LIN {X 0,Y 418.229,Z 234.888,A -85,B 0,C 180,E1 -10045.167,E2 -10045.167} C_VEL
LIN {X 0,Y 418.217,Z 234.887,A -85,B 0,C 180,E1 -10047.48,E2 -10047.48} C_VEL
LIN {X 0,Y 418.245,Z 234.887,A -85,B 0,C 180,E1 -10050.903,E2 -10050.903} C_VEL
LIN {X 0,Y 418.249,Z 234.881,A -85,B 0,C 180,E1 -10054.103,E2 -10054.103} C_VEL
LIN {X 0,Y 418.216,Z 234.893,A -85,B 0,C 180,E1 -10057.271,E2 -10057.271} C_VEL
LIN {X 0,Y 418.27,Z 234.878,A -85,B 0,C 180,E1 -10060.372,E2 -10060.372} C_VEL
LIN {X 0,Y 418.307,Z 234.881,A -85,B 0,C 180,E1 -10063.412,E2 -10063.412} C_VEL
LIN {X 0,Y 418.341,Z 234.871,A -85,B 0,C 180,E1 -10067.007,E2 -10067.007} C_VEL
LIN {X 0,Y 418.335,Z 234.872,A -85,B 0,C 180,E1 -10070.336,E2 -10070.336} C_VEL
LIN {X 0,Y 418.445,Z 234.858,A -85,B 0,C 180,E1 -10073.255,E2 -10073.255} C_VEL
LIN {X 0,Y 418.328,Z 234.872,A -85,B 0,C 180,E1 -10075.188,E2 -10075.188} C_VEL
LIN {X 0,Y 418.543,Z 234.852,A -85,B 0,C 180,E1 -10078.082,E2 -10078.082} C_VEL
LIN {X 0,Y 418.47,Z 234.854,A -85,B 0,C 180,E1 -10080.969,E2 -10080.969} C_VEL
LIN {X 0,Y 418.477,Z 234.853,A -85,B 0,C 180,E1 -10082.894,E2 -10082.894} C_VEL
LIN {X 0,Y 418.494,Z 234.853,A -85,B 0,C 180,E1 -10085.789,E2 -10085.789} C_VEL
LIN {X 0,Y 418.38,Z 234.868,A -85,B 0,C 180,E1 -10088.701,E2 -10088.701} C_VEL
LIN {X 0,Y 418.324,Z 234.872,A -85,B 0,C 180,E1 -10091.636,E2 -10091.636} C_VEL
LIN {X 0,Y 418.315,Z 234.881,A -85,B 0,C 180,E1 -10094.602,E2 -10094.602} C_VEL
LIN {X 0,Y 418.296,Z 234.875,A -85,B 0,C 180,E1 -10097.609,E2 -10097.609} C_VEL
LIN {X 0,Y 418.267,Z 234.886,A -85,B 0,C 180,E1 -10100.667,E2 -10100.667} C_VEL
LIN {X 0,Y 418.276,Z 234.878,A -85,B 0,C 180,E1 -10103.787,E2 -10103.787} C_VEL
LIN {X 0,Y 418.227,Z 234.891,A -85,B 0,C 180,E1 -10107.046,E2 -10107.046} C_VEL
LIN {X 0,Y 418.259,Z 234.88,A -85,B 0,C 180,E1 -10110.276,E2 -10110.276} C_VEL
LIN {X 0,Y 418.253,Z 234.883,A -85,B 0,C 180,E1 -10113.682,E2 -10113.682} C_VEL
LIN {X 0,Y 418.259,Z 234.887,A -85,B 0,C 180,E1 -10117.227,E2 -10117.227} C_VEL
LIN {X 0,Y 418.229,Z 234.885,A -85,B 0,C 180,E1 -10120.869,E2 -10120.869} C_VEL
LIN {X 0,Y 418.202,Z 234.893,A -85,B 0,C 180,E1 -10123.727,E2 -10123.727} C_VEL
LIN {X 0,Y 418.207,Z 234.887,A -85,B 0,C 180,E1 -10126.447,E2 -10126.447} C_VEL
LIN {X 0,Y 418.228,Z 234.885,A -85,B 0,C 180,E1 -10129.134,E2 -10129.134} C_VEL
LIN {X 0,Y 418.255,Z 234.88,A -85,B 0,C 180,E1 -10132.776,E2 -10132.776} C_VEL
LIN {X 0,Y 418.258,Z 234.884,A -85,B 0,C 180,E1 -10136.322,E2 -10136.322} C_VEL
LIN {X 0,Y 418.261,Z 234.883,A -85,B 0,C 180,E1 -10139.728,E2 -10139.728} C_VEL
LIN {X 0,Y 418.285,Z 234.885,A -85,B 0,C 180,E1 -10143.29,E2 -10143.29} C_VEL
LIN {X 0,Y 418.328,Z 235.082,A -85,B 0,C 180,E1 -10143.562,E2 -10143.562} C_VEL
LIN {X 0,Y 420.651,Z 247.12,A -85,B 0,C 180,E1 -10146.359,E2 -10146.359} C_VEL
LIN {X 0,Y 420.968,Z 250.295,A -85,B 0,C 180,E1 -10147.061,E2 -10147.061} C_VEL
LIN {X 0,Y 419.806,Z 267.603,A -85,B 0,C 180,E1 -10150.691,E2 -10150.691} C_VEL
LIN {X 0,Y 419.723,Z 269.608,A -85,B 0,C 180,E1 -10151.068,E2 -10151.068} C_VEL
LIN {X 0,Y 421.486,Z 280.526,A -85,B 0,C 180,E1 -10151.383,E2 -10151.383} C_VEL
LIN {X 0,Y 423.53,Z 293.837,A -85,B 0,C 180,E1 -10151.714,E2 -10151.714} C_VEL
LIN {X 0,Y 422.409,Z 377.431,A -85,B 0,C 180,E1 -10153.227,E2 -10153.227} C_VEL
LIN {X 0,Y 422.039,Z 390.51,A -85,B 0,C 180,E1 -10153.647,E2 -10153.647} C_VEL
LIN {X 0,Y 421.453,Z 402.615,A -85,B 0,C 180,E1 -10154.214,E2 -10154.214} C_VEL
LIN {X 0,Y 420.729,Z 414.885,A -85,B 0,C 180,E1 -10154.993,E2 -10154.993} C_VEL
LIN {X 0,Y 419.97,Z 427.124,A -85,B 0,C 180,E1 -10156.014,E2 -10156.014} C_VEL
LIN {X 0,Y 419.288,Z 438.018,A -85,B 0,C 180,E1 -10157.166,E2 -10157.166} C_VEL
LIN {X 0,Y 418.646,Z 447.21,A -85,B 0,C 180,E1 -10158.377,E2 -10158.377} C_VEL
LIN {X 0,Y 418.062,Z 456.167,A -85,B 0,C 180,E1 -10159.832,E2 -10159.832} C_VEL
LIN {X 0,Y 417.663,Z 463.349,A -85,B 0,C 180,E1 -10161.288,E2 -10161.288} C_VEL
LIN {X 0,Y 417.306,Z 469.059,A -85,B 0,C 180,E1 -10162.742,E2 -10162.742} C_VEL
LIN {X 0,Y 417.136,Z 473.548,A -85,B 0,C 180,E1 -10164.197,E2 -10164.197} C_VEL
LIN {X 0,Y 417.122,Z 475.915,A -85,B 0,C 180,E1 -10165.166,E2 -10165.166} C_VEL
LIN {X 0,Y 417.006,Z 477.844,A -85,B 0,C 180,E1 -10166.133,E2 -10166.133} C_VEL
LIN {X 0,Y 416.99,Z 479.33,A -85,B 0,C 180,E1 -10167.1,E2 -10167.1} C_VEL
LIN {X 0,Y 417.037,Z 480.372,A -85,B 0,C 180,E1 -10168.067,E2 -10168.067} C_VEL
LIN {X 0,Y 416.999,Z 481.017,A -85,B 0,C 180,E1 -10169.033,E2 -10169.033} C_VEL
LIN {X 0,Y 416.989,Z 481.272,A -85,B 0,C 180,E1 -10169.998,E2 -10169.998} C_VEL
LIN {X 0,Y 416.999,Z 481.107,A -85,B 0,C 180,E1 -10170.964,E2 -10170.964} C_VEL
LIN {X 0,Y 417.036,Z 480.518,A -85,B 0,C 180,E1 -10171.93,E2 -10171.93} C_VEL
LIN {X 0,Y 417.005,Z 478.156,A -85,B 0,C 180,E1 -10173.864,E2 -10173.864} C_VEL
LIN {X 0,Y 417.163,Z 475.238,A -85,B 0,C 180,E1 -10175.315,E2 -10175.315} C_VEL
LIN {X 0,Y 417.255,Z 471.278,A -85,B 0,C 180,E1 -10176.769,E2 -10176.769} C_VEL
LIN {X 0,Y 417.612,Z 465.193,A -85,B 0,C 180,E1 -10178.466,E2 -10178.466} C_VEL
LIN {X 0,Y 418.022,Z 458.52,A -85,B 0,C 180,E1 -10179.921,E2 -10179.921} C_VEL
LIN {X 0,Y 418.596,Z 450.239,A -85,B 0,C 180,E1 -10181.376,E2 -10181.376} C_VEL
LIN {X 0,Y 419.307,Z 441.768,A -85,B 0,C 180,E1 -10182.583,E2 -10182.583} C_VEL
LIN {X 0,Y 420.041,Z 431.587,A -85,B 0,C 180,E1 -10183.763,E2 -10183.763} C_VEL
LIN {X 0,Y 420.683,Z 420.983,A -85,B 0,C 180,E1 -10184.758,E2 -10184.758} C_VEL
LIN {X 0,Y 421.436,Z 409.695,A -85,B 0,C 180,E1 -10185.597,E2 -10185.597} C_VEL
LIN {X 0,Y 422.138,Z 398.235,A -85,B 0,C 180,E1 -10186.253,E2 -10186.253} C_VEL
LIN {X 0,Y 422.668,Z 385.205,A -85,B 0,C 180,E1 -10186.791,E2 -10186.791} C_VEL
LIN {X 0,Y 423.061,Z 372.908,A -85,B 0,C 180,E1 -10187.117,E2 -10187.117} C_VEL
LIN {X 0,Y 424.16,Z 293.421,A -85,B 0,C 180,E1 -10188.564,E2 -10188.564} C_VEL
LIN {X 0,Y 419.995,Z 269.208,A -85,B 0,C 180,E1 -10189.255,E2 -10189.255} C_VEL
LIN {X 0,Y 420.004,Z 267.48,A -85,B 0,C 180,E1 -10189.55,E2 -10189.55} C_VEL
LIN {X 0,Y 421.06,Z 250.814,A -85,B 0,C 180,E1 -10192.955,E2 -10192.955} C_VEL
LIN {X 0,Y 420.401,Z 245.236,A -85,B 0,C 180,E1 -10194.176,E2 -10194.176} C_VEL
LIN {X 0,Y 418.317,Z 234.989,A -85,B 0,C 180,E1 -10196.569,E2 -10196.569} C_VEL
LIN {X 0,Y 418.275,Z 234.882,A -85,B 0,C 180,E1 -10199.159,E2 -10199.159} C_VEL
LIN {X 0,Y 418.266,Z 234.883,A -85,B 0,C 180,E1 -10202.84,E2 -10202.84} C_VEL
LIN {X 0,Y 418.251,Z 234.888,A -85,B 0,C 180,E1 -10206.234,E2 -10206.234} C_VEL
LIN {X 0,Y 418.206,Z 234.891,A -85,B 0,C 180,E1 -10209.684,E2 -10209.684} C_VEL
LIN {X 0,Y 418.214,Z 234.891,A -85,B 0,C 180,E1 -10212.314,E2 -10212.314} C_VEL
LIN {X 0,Y 418.239,Z 234.883,A -85,B 0,C 180,E1 -10215.104,E2 -10215.104} C_VEL
LIN {X 0,Y 418.222,Z 234.889,A -85,B 0,C 180,E1 -10217.76,E2 -10217.76} C_VEL
LIN {X 0,Y 418.236,Z 234.884,A -85,B 0,C 180,E1 -10221.551,E2 -10221.551} C_VEL
LIN {X 0,Y 418.25,Z 234.884,A -85,B 0,C 180,E1 -10225.153,E2 -10225.153} C_VEL
LIN {X 0,Y 418.244,Z 234.882,A -85,B 0,C 180,E1 -10227.467,E2 -10227.467} C_VEL
LIN {X 0,Y 418.259,Z 234.885,A -85,B 0,C 180,E1 -10230.893,E2 -10230.893} C_VEL
LIN {X 0,Y 418.215,Z 234.883,A -85,B 0,C 180,E1 -10234.087,E2 -10234.087} C_VEL
LIN {X 0,Y 418.221,Z 234.885,A -85,B 0,C 180,E1 -10237.258,E2 -10237.258} C_VEL
LIN {X 0,Y 418.245,Z 234.885,A -85,B 0,C 180,E1 -10240.357,E2 -10240.357} C_VEL
LIN {X 0,Y 418.273,Z 234.879,A -85,B 0,C 180,E1 -10243.397,E2 -10243.397} C_VEL
LIN {X 0,Y 418.337,Z 234.874,A -85,B 0,C 180,E1 -10246.994,E2 -10246.994} C_VEL
LIN {X 0,Y 418.316,Z 234.875,A -85,B 0,C 180,E1 -10250.322,E2 -10250.322} C_VEL
LIN {X 0,Y 418.452,Z 234.861,A -85,B 0,C 180,E1 -10253.242,E2 -10253.242} C_VEL
LIN {X 0,Y 418.306,Z 234.879,A -85,B 0,C 180,E1 -10255.175,E2 -10255.175} C_VEL
LIN {X 0,Y 418.518,Z 234.85,A -85,B 0,C 180,E1 -10258.069,E2 -10258.069} C_VEL
LIN {X 0,Y 418.649,Z 234.832,A -85,B 0,C 180,E1 -10259.994,E2 -10259.994} C_VEL
LIN {X 0,Y 418.48,Z 234.855,A -85,B 0,C 180,E1 -10262.881,E2 -10262.881} C_VEL
LIN {X 0,Y 418.439,Z 234.86,A -85,B 0,C 180,E1 -10266.474,E2 -10266.474} C_VEL
LIN {X 0,Y 418.372,Z 234.869,A -85,B 0,C 180,E1 -10268.689,E2 -10268.689} C_VEL
LIN {X 0,Y 418.307,Z 234.881,A -85,B 0,C 180,E1 -10271.624,E2 -10271.624} C_VEL
LIN {X 0,Y 418.279,Z 234.881,A -85,B 0,C 180,E1 -10274.59,E2 -10274.59} C_VEL
LIN {X 0,Y 418.255,Z 234.884,A -85,B 0,C 180,E1 -10277.597,E2 -10277.597} C_VEL
LIN {X 0,Y 418.244,Z 234.886,A -85,B 0,C 180,E1 -10280.655,E2 -10280.655} C_VEL
LIN {X 0,Y 418.345,Z 235.06,A -85,B 0,C 180,E1 -10281.902,E2 -10281.902} C_VEL
LIN {X 0,Y 420.612,Z 246.343,A -85,B 0,C 180,E1 -10284.419,E2 -10284.419} C_VEL
LIN {X 0,Y 420.097,Z 258.242,A -85,B 0,C 180,E1 -10286.776,E2 -10286.776} C_VEL
LIN {X 0,Y 424.106,Z 279.087,A -85,B 0,C 180,E1 -10287.408,E2 -10287.408} C_VEL
LIN {X 0,Y 424.207,Z 285.864,A -85,B 0,C 180,E1 -10287.544,E2 -10287.544} C_VEL
LIN {X 0,Y 422.969,Z 366.776,A -85,B 0,C 180,E1 -10289.036,E2 -10289.036} C_VEL
LIN {X 0,Y 422.459,Z 380.788,A -85,B 0,C 180,E1 -10289.501,E2 -10289.501} C_VEL
LIN {X 0,Y 421.952,Z 393.509,A -85,B 0,C 180,E1 -10290.137,E2 -10290.137} C_VEL
LIN {X 0,Y 421.204,Z 406.059,A -85,B 0,C 180,E1 -10290.985,E2 -10290.985} C_VEL
LIN {X 0,Y 420.487,Z 416.903,A -85,B 0,C 180,E1 -10291.925,E2 -10291.925} C_VEL
LIN {X 0,Y 419.791,Z 426.126,A -85,B 0,C 180,E1 -10292.911,E2 -10292.911} C_VEL
LIN {X 0,Y 419.091,Z 435.683,A -85,B 0,C 180,E1 -10294.169,E2 -10294.169} C_VEL
LIN {X 0,Y 418.485,Z 443.34,A -85,B 0,C 180,E1 -10295.397,E2 -10295.397} C_VEL
LIN {X 0,Y 417.912,Z 451.314,A -85,B 0,C 180,E1 -10296.978,E2 -10296.978} C_VEL
LIN {X 0,Y 417.525,Z 457.387,A -85,B 0,C 180,E1 -10298.51,E2 -10298.51} C_VEL
LIN {X 0,Y 417.217,Z 462.602,A -85,B 0,C 180,E1 -10300.241,E2 -10300.241} C_VEL
LIN {X 0,Y 417.03,Z 465.647,A -85,B 0,C 180,E1 -10301.601,E2 -10301.601} C_VEL
LIN {X 0,Y 416.878,Z 468.506,A -85,B 0,C 180,E1 -10303.541,E2 -10303.541} C_VEL
LIN {X 0,Y 416.845,Z 469.573,A -85,B 0,C 180,E1 -10305.069,E2 -10305.069} C_VEL
LIN {X 0,Y 416.8,Z 469.657,A -85,B 0,C 180,E1 -10306.46,E2 -10306.46} C_VEL
LIN {X 0,Y 416.838,Z 468.894,A -85,B 0,C 180,E1 -10307.875,E2 -10307.875} C_VEL
LIN {X 0,Y 416.91,Z 467.21,A -85,B 0,C 180,E1 -10309.325,E2 -10309.325} C_VEL
LIN {X 0,Y 417.058,Z 464.506,A -85,B 0,C 180,E1 -10310.805,E2 -10310.805} C_VEL
LIN {X 0,Y 417.231,Z 460.612,A -85,B 0,C 180,E1 -10312.328,E2 -10312.328} C_VEL
LIN {X 0,Y 417.543,Z 455.256,A -85,B 0,C 180,E1 -10313.909,E2 -10313.909} C_VEL
LIN {X 0,Y 418.018,Z 448.556,A -85,B 0,C 180,E1 -10315.452,E2 -10315.452} C_VEL
LIN {X 0,Y 418.492,Z 440.342,A -85,B 0,C 180,E1 -10316.945,E2 -10316.945} C_VEL
LIN {X 0,Y 419.13,Z 431.379,A -85,B 0,C 180,E1 -10318.26,E2 -10318.26} C_VEL
LIN {X 0,Y 419.746,Z 421.55,A -85,B 0,C 180,E1 -10319.433,E2 -10319.433} C_VEL
LIN {X 0,Y 420.458,Z 410.995,A -85,B 0,C 180,E1 -10320.441,E2 -10320.441} C_VEL
LIN {X 0,Y 421.146,Z 398.632,A -85,B 0,C 180,E1 -10321.375,E2 -10321.375} C_VEL
LIN {X 0,Y 421.714,Z 387.532,A -85,B 0,C 180,E1 -10322.017,E2 -10322.017} C_VEL
LIN {X 0,Y 422.155,Z 374.294,A -85,B 0,C 180,E1 -10322.571,E2 -10322.571} C_VEL
LIN {X 0,Y 422.52,Z 360.472,A -85,B 0,C 180,E1 -10322.932,E2 -10322.932} C_VEL
LIN {X 0,Y 423.47,Z 279.209,A -85,B 0,C 180,E1 -10324.385,E2 -10324.385} C_VEL
LIN {X 0,Y 420.91,Z 264.799,A -85,B 0,C 180,E1 -10324.759,E2 -10324.759} C_VEL
LIN {X 0,Y 419.872,Z 261.526,A -85,B 0,C 180,E1 -10324.945,E2 -10324.945} C_VEL
LIN {X 0,Y 418.385,Z 258.162,A -85,B 0,C 180,E1 -10325.342,E2 -10325.342} C_VEL
LIN {X 0,Y 416.377,Z 254.492,A -85,B 0,C 180,E1 -10326.065,E2 -10326.065} C_VEL
LIN {X 0,Y 413.702,Z 248.584,A -85,B 0,C 180,E1 -10327.592,E2 -10327.592} C_VEL
LIN {X 0,Y 413.252,Z 246.492,A -85,B 0,C 180,E1 -10328.11,E2 -10328.11} C_VEL
LIN {X 0,Y 411.256,Z 235.918,A -85,B 0,C 180,E1 -10330.796,E2 -10330.796} C_VEL
LIN {X 0,Y 411.199,Z 235.765,A -85,B 0,C 180,E1 -10334.132,E2 -10334.132} C_VEL
LIN {X 0,Y 411.242,Z 235.755,A -85,B 0,C 180,E1 -10337.166,E2 -10337.166} C_VEL
LIN {X 0,Y 411.237,Z 235.757,A -85,B 0,C 180,E1 -10340.162,E2 -10340.162} C_VEL
LIN {X 0,Y 411.386,Z 235.739,A -85,B 0,C 180,E1 -10343.134,E2 -10343.134} C_VEL
LIN {X 0,Y 411.249,Z 235.758,A -85,B 0,C 180,E1 -10345.1,E2 -10345.1} C_VEL
LIN {X 0,Y 411.441,Z 235.729,A -85,B 0,C 180,E1 -10348.044,E2 -10348.044} C_VEL
LIN {X 0,Y 411.569,Z 235.713,A -85,B 0,C 180,E1 -10350.002,E2 -10350.002} C_VEL
LIN {X 0,Y 411.403,Z 235.74,A -85,B 0,C 180,E1 -10352.939,E2 -10352.939} C_VEL
LIN {X 0,Y 411.419,Z 235.733,A -85,B 0,C 180,E1 -10355.884,E2 -10355.884} C_VEL
LIN {X 0,Y 411.287,Z 235.751,A -85,B 0,C 180,E1 -10358.848,E2 -10358.848} C_VEL
LIN {X 0,Y 411.233,Z 235.758,A -85,B 0,C 180,E1 -10361.836,E2 -10361.836} C_VEL
LIN {X 0,Y 411.197,Z 235.761,A -85,B 0,C 180,E1 -10364.857,E2 -10364.857} C_VEL
LIN {X 0,Y 411.184,Z 235.765,A -85,B 0,C 180,E1 -10367.92,E2 -10367.92} C_VEL
LIN {X 0,Y 411.13,Z 235.769,A -85,B 0,C 180,E1 -10371.039,E2 -10371.039} C_VEL
LIN {X 0,Y 411.165,Z 235.767,A -85,B 0,C 180,E1 -10374.221,E2 -10374.221} C_VEL
LIN {X 0,Y 411.201,Z 235.762,A -85,B 0,C 180,E1 -10377.483,E2 -10377.483} C_VEL
LIN {X 0,Y 411.144,Z 235.767,A -85,B 0,C 180,E1 -10380.853,E2 -10380.853} C_VEL
LIN {X 0,Y 411.153,Z 235.771,A -85,B 0,C 180,E1 -10384.34,E2 -10384.34} C_VEL
LIN {X 0,Y 411.153,Z 235.769,A -85,B 0,C 180,E1 -10387.98,E2 -10387.98} C_VEL
LIN {X 0,Y 411.164,Z 235.764,A -85,B 0,C 180,E1 -10391.243,E2 -10391.243} C_VEL
LIN {X 0,Y 411.19,Z 235.768,A -85,B 0,C 180,E1 -10394.49,E2 -10394.49} C_VEL
LIN {X 0,Y 411.193,Z 235.761,A -85,B 0,C 180,E1 -10397.304,E2 -10397.304} C_VEL
LIN {X 0,Y 411.196,Z 235.767,A -85,B 0,C 180,E1 -10400.785,E2 -10400.785} C_VEL
LIN {X 0,Y 411.168,Z 235.766,A -85,B 0,C 180,E1 -10404.479,E2 -10404.479} C_VEL
LIN {X 0,Y 411.179,Z 235.769,A -85,B 0,C 180,E1 -10406.881,E2 -10406.881} C_VEL
LIN {X 0,Y 411.192,Z 235.763,A -85,B 0,C 180,E1 -10410.656,E2 -10410.656} C_VEL
LIN {X 0,Y 411.217,Z 235.76,A -85,B 0,C 180,E1 -10413.627,E2 -10413.627} C_VEL
LIN {X 0,Y 411.18,Z 235.765,A -85,B 0,C 180,E1 -10416.86,E2 -10416.86} C_VEL
LIN {X 0,Y 411.201,Z 235.76,A -85,B 0,C 180,E1 -10420.059,E2 -10420.059} C_VEL
LIN {X 0,Y 411.254,Z 235.756,A -85,B 0,C 180,E1 -10423.139,E2 -10423.139} C_VEL
LIN {X 0,Y 411.3,Z 235.747,A -85,B 0,C 180,E1 -10426.904,E2 -10426.904} C_VEL
LIN {X 0,Y 411.288,Z 235.751,A -85,B 0,C 180,E1 -10430.168,E2 -10430.168} C_VEL
LIN {X 0,Y 411.393,Z 235.736,A -85,B 0,C 180,E1 -10433.139,E2 -10433.139} C_VEL
LIN {X 0,Y 411.299,Z 235.747,A -85,B 0,C 180,E1 -10435.106,E2 -10435.106} C_VEL
LIN {X 0,Y 411.512,Z 235.728,A -85,B 0,C 180,E1 -10438.049,E2 -10438.049} C_VEL
LIN {X 0,Y 411.435,Z 235.73,A -85,B 0,C 180,E1 -10440.985,E2 -10440.985} C_VEL
LIN {X 0,Y 411.436,Z 235.73,A -85,B 0,C 180,E1 -10442.944,E2 -10442.944} C_VEL
LIN {X 0,Y 411.439,Z 235.733,A -85,B 0,C 180,E1 -10445.889,E2 -10445.889} C_VEL
LIN {X 0,Y 411.321,Z 235.746,A -85,B 0,C 180,E1 -10448.852,E2 -10448.852} C_VEL
LIN {X 0,Y 411.294,Z 235.749,A -85,B 0,C 180,E1 -10451.838,E2 -10451.838} C_VEL
LIN {X 0,Y 411.273,Z 235.754,A -85,B 0,C 180,E1 -10454.858,E2 -10454.858} C_VEL
LIN {X 0,Y 411.262,Z 235.752,A -85,B 0,C 180,E1 -10457.92,E2 -10457.92} C_VEL
LIN {X 0,Y 411.214,Z 235.762,A -85,B 0,C 180,E1 -10461.038,E2 -10461.038} C_VEL
LIN {X 0,Y 411.21,Z 235.759,A -85,B 0,C 180,E1 -10464.222,E2 -10464.222} C_VEL
LIN {X 0,Y 411.166,Z 235.766,A -85,B 0,C 180,E1 -10467.49,E2 -10467.49} C_VEL
LIN {X 0,Y 411.216,Z 235.758,A -85,B 0,C 180,E1 -10469.717,E2 -10469.717} C_VEL
LIN {X 0,Y 411.226,Z 235.764,A -85,B 0,C 180,E1 -10473.159,E2 -10473.159} C_VEL
LIN {X 0,Y 411.213,Z 235.758,A -85,B 0,C 180,E1 -10476.555,E2 -10476.555} C_VEL
LIN {X 0,Y 411.191,Z 235.764,A -85,B 0,C 180,E1 -10479.722,E2 -10479.722} C_VEL
LIN {X 0,Y 411.14,Z 235.77,A -85,B 0,C 180,E1 -10483.143,E2 -10483.143} C_VEL
LIN {X 0,Y 411.177,Z 235.767,A -85,B 0,C 180,E1 -10485.885,E2 -10485.885} C_VEL
LIN {X 0,Y 411.179,Z 235.766,A -85,B 0,C 180,E1 -10489.494,E2 -10489.494} C_VEL
LIN {X 0,Y 411.203,Z 235.764,A -85,B 0,C 180,E1 -10492.026,E2 -10492.026} C_VEL
LIN {X 0,Y 411.219,Z 235.761,A -85,B 0,C 180,E1 -10495.666,E2 -10495.666} C_VEL
LIN {X 0,Y 411.209,Z 235.759,A -85,B 0,C 180,E1 -10499.153,E2 -10499.153} C_VEL
LIN {X 0,Y 411.209,Z 235.766,A -85,B 0,C 180,E1 -10502.517,E2 -10502.517} C_VEL
LIN {X 0,Y 411.259,Z 235.867,A -85,B 0,C 180,E1 -10503.286,E2 -10503.286} C_VEL
LIN {X 0,Y 413.416,Z 246.889,A -85,B 0,C 180,E1 -10505.92,E2 -10505.92} C_VEL
LIN {X 0,Y 413.979,Z 251.745,A -85,B 0,C 180,E1 -10507.015,E2 -10507.015} C_VEL
LIN {X 0,Y 412.791,Z 269.292,A -85,B 0,C 180,E1 -10510.738,E2 -10510.738} C_VEL
LIN {X 0,Y 413.105,Z 272.049,A -85,B 0,C 180,E1 -10510.869,E2 -10510.869} C_VEL
LIN {X 0,Y 416.732,Z 294.503,A -85,B 0,C 180,E1 -10511.448,E2 -10511.448} C_VEL
LIN {X 0,Y 415.576,Z 377.319,A -85,B 0,C 180,E1 -10512.974,E2 -10512.974} C_VEL
LIN {X 0,Y 415.108,Z 391.143,A -85,B 0,C 180,E1 -10513.429,E2 -10513.429} C_VEL
LIN {X 0,Y 414.551,Z 403.062,A -85,B 0,C 180,E1 -10514.007,E2 -10514.007} C_VEL
LIN {X 0,Y 413.841,Z 414.374,A -85,B 0,C 180,E1 -10514.737,E2 -10514.737} C_VEL
LIN {X 0,Y 413.179,Z 425.156,A -85,B 0,C 180,E1 -10515.631,E2 -10515.631} C_VEL
LIN {X 0,Y 412.383,Z 436.605,A -85,B 0,C 180,E1 -10516.823,E2 -10516.823} C_VEL
LIN {X 0,Y 411.789,Z 445.213,A -85,B 0,C 180,E1 -10517.931,E2 -10517.931} C_VEL
LIN {X 0,Y 411.182,Z 453.143,A -85,B 0,C 180,E1 -10519.162,E2 -10519.162} C_VEL
LIN {X 0,Y 410.696,Z 460.873,A -85,B 0,C 180,E1 -10520.642,E2 -10520.642} C_VEL
LIN {X 0,Y 410.363,Z 467.076,A -85,B 0,C 180,E1 -10522.124,E2 -10522.124} C_VEL
LIN {X 0,Y 410.108,Z 472.311,A -85,B 0,C 180,E1 -10523.713,E2 -10523.713} C_VEL
LIN {X 0,Y 410.036,Z 475.758,A -85,B 0,C 180,E1 -10525.082,E2 -10525.082} C_VEL
LIN {X 0,Y 409.926,Z 477.698,A -85,B 0,C 180,E1 -10526.066,E2 -10526.066} C_VEL
LIN {X 0,Y 409.888,Z 479.202,A -85,B 0,C 180,E1 -10527.05,E2 -10527.05} C_VEL
LIN {X 0,Y 409.933,Z 480.252,A -85,B 0,C 180,E1 -10528.033,E2 -10528.033} C_VEL
LIN {X 0,Y 409.926,Z 480.907,A -85,B 0,C 180,E1 -10529.016,E2 -10529.016} C_VEL
LIN {X 0,Y 409.913,Z 481.169,A -85,B 0,C 180,E1 -10529.998,E2 -10529.998} C_VEL
LIN {X 0,Y 409.925,Z 481.02,A -85,B 0,C 180,E1 -10530.981,E2 -10530.981} C_VEL
LIN {X 0,Y 409.933,Z 480.438,A -85,B 0,C 180,E1 -10531.963,E2 -10531.963} C_VEL
LIN {X 0,Y 409.927,Z 478.088,A -85,B 0,C 180,E1 -10533.931,E2 -10533.931} C_VEL
LIN {X 0,Y 410.081,Z 475.183,A -85,B 0,C 180,E1 -10535.407,E2 -10535.407} C_VEL
LIN {X 0,Y 410.193,Z 471.236,A -85,B 0,C 180,E1 -10536.886,E2 -10536.886} C_VEL
LIN {X 0,Y 410.498,Z 466.147,A -85,B 0,C 180,E1 -10538.366,E2 -10538.366} C_VEL
LIN {X 0,Y 410.914,Z 459.751,A -85,B 0,C 180,E1 -10539.846,E2 -10539.846} C_VEL
LIN {X 0,Y 411.502,Z 451.742,A -85,B 0,C 180,E1 -10541.325,E2 -10541.325} C_VEL
LIN {X 0,Y 412.385,Z 441.792,A -85,B 0,C 180,E1 -10542.798,E2 -10542.798} C_VEL
LIN {X 0,Y 413.103,Z 432.283,A -85,B 0,C 180,E1 -10543.931,E2 -10543.931} C_VEL
LIN {X 0,Y 413.83,Z 421.097,A -85,B 0,C 180,E1 -10545.008,E2 -10545.008} C_VEL
LIN {X 0,Y 414.62,Z 409.885,A -85,B 0,C 180,E1 -10545.86,E2 -10545.86} C_VEL
LIN {X 0,Y 415.359,Z 398.557,A -85,B 0,C 180,E1 -10546.525,E2 -10546.525} C_VEL
LIN {X 0,Y 415.908,Z 385.789,A -85,B 0,C 180,E1 -10547.072,E2 -10547.072} C_VEL
LIN {X 0,Y 416.371,Z 372.533,A -85,B 0,C 180,E1 -10547.432,E2 -10547.432} C_VEL
LIN {X 0,Y 417.434,Z 293.78,A -85,B 0,C 180,E1 -10548.898,E2 -10548.898} C_VEL
LIN {X 0,Y 413.326,Z 270.34,A -85,B 0,C 180,E1 -10549.575,E2 -10549.575} C_VEL
LIN {X 0,Y 413.082,Z 268.6,A -85,B 0,C 180,E1 -10549.678,E2 -10549.678} C_VEL
LIN {X 0,Y 414.121,Z 252.699,A -85,B 0,C 180,E1 -10552.973,E2 -10552.973} C_VEL
LIN {X 0,Y 413.941,Z 249.262,A -85,B 0,C 180,E1 -10553.722,E2 -10553.722} C_VEL
LIN {X 0,Y 411.965,Z 239.075,A -85,B 0,C 180,E1 -10556.072,E2 -10556.072} C_VEL
LIN {X 0,Y 411.251,Z 235.81,A -85,B 0,C 180,E1 -10556.917,E2 -10556.917} C_VEL
LIN {X 0,Y 411.21,Z 235.765,A -85,B 0,C 180,E1 -10559.71,E2 -10559.71} C_VEL
LIN {X 0,Y 411.216,Z 235.762,A -85,B 0,C 180,E1 -10563.152,E2 -10563.152} C_VEL
LIN {X 0,Y 411.199,Z 235.764,A -85,B 0,C 180,E1 -10566.548,E2 -10566.548} C_VEL
LIN {X 0,Y 411.175,Z 235.767,A -85,B 0,C 180,E1 -10569.716,E2 -10569.716} C_VEL
LIN {X 0,Y 411.168,Z 235.764,A -85,B 0,C 180,E1 -10573.131,E2 -10573.131} C_VEL
LIN {X 0,Y 411.168,Z 235.766,A -85,B 0,C 180,E1 -10575.878,E2 -10575.878} C_VEL
LIN {X 0,Y 411.161,Z 235.767,A -85,B 0,C 180,E1 -10579.488,E2 -10579.488} C_VEL
LIN {X 0,Y 411.183,Z 235.766,A -85,B 0,C 180,E1 -10582.02,E2 -10582.02} C_VEL
LIN {X 0,Y 411.202,Z 235.762,A -85,B 0,C 180,E1 -10585.119,E2 -10585.119} C_VEL
LIN {X 0,Y 411.164,Z 235.766,A -85,B 0,C 180,E1 -10587.998,E2 -10587.998} C_VEL
LIN {X 0,Y 411.171,Z 235.765,A -85,B 0,C 180,E1 -10591.401,E2 -10591.401} C_VEL
LIN {X 0,Y 411.186,Z 235.767,A -85,B 0,C 180,E1 -10594.936,E2 -10594.936} C_VEL
LIN {X 0,Y 411.195,Z 235.759,A -85,B 0,C 180,E1 -10597.908,E2 -10597.908} C_VEL
LIN {X 0,Y 411.177,Z 235.764,A -85,B 0,C 180,E1 -10601.044,E2 -10601.044} C_VEL
LIN {X 0,Y 411.199,Z 235.759,A -85,B 0,C 180,E1 -10604.124,E2 -10604.124} C_VEL
LIN {X 0,Y 411.294,Z 235.749,A -85,B 0,C 180,E1 -10607.16,E2 -10607.16} C_VEL
LIN {X 0,Y 411.27,Z 235.753,A -85,B 0,C 180,E1 -10610.155,E2 -10610.155} C_VEL
LIN {X 0,Y 411.418,Z 235.738,A -85,B 0,C 180,E1 -10613.126,E2 -10613.126} C_VEL
LIN {X 0,Y 411.279,Z 235.753,A -85,B 0,C 180,E1 -10615.093,E2 -10615.093} C_VEL
LIN {X 0,Y 411.487,Z 235.726,A -85,B 0,C 180,E1 -10618.036,E2 -10618.036} C_VEL
LIN {X 0,Y 411.619,Z 235.708,A -85,B 0,C 180,E1 -10619.994,E2 -10619.994} C_VEL
LIN {X 0,Y 411.437,Z 235.732,A -85,B 0,C 180,E1 -10622.931,E2 -10622.931} C_VEL
LIN {X 0,Y 411.407,Z 235.738,A -85,B 0,C 180,E1 -10626.861,E2 -10626.861} C_VEL
LIN {X 0,Y 411.283,Z 235.755,A -85,B 0,C 180,E1 -10629.832,E2 -10629.832} C_VEL
LIN {X 0,Y 411.286,Z 235.754,A -85,B 0,C 180,E1 -10633.103,E2 -10633.103} C_VEL
LIN {X 0,Y 411.225,Z 235.761,A -85,B 0,C 180,E1 -10636.882,E2 -10636.882} C_VEL
LIN {X 0,Y 411.221,Z 235.764,A -85,B 0,C 180,E1 -10639.979,E2 -10639.979} C_VEL
LIN {X 0,Y 411.254,Z 235.868,A -85,B 0,C 180,E1 -10641.548,E2 -10641.548} C_VEL
LIN {X 0,Y 413.129,Z 244.487,A -85,B 0,C 180,E1 -10643.555,E2 -10643.555} C_VEL
LIN {X 0,Y 413.734,Z 247.939,A -85,B 0,C 180,E1 -10644.317,E2 -10644.317} C_VEL
LIN {X 0,Y 413.234,Z 258.335,A -85,B 0,C 180,E1 -10646.404,E2 -10646.404} C_VEL
LIN {X 0,Y 417.379,Z 279.278,A -85,B 0,C 180,E1 -10647.066,E2 -10647.066} C_VEL
LIN {X 0,Y 417.607,Z 283.906,A -85,B 0,C 180,E1 -10647.169,E2 -10647.169} C_VEL
LIN {X 0,Y 416.24,Z 367.025,A -85,B 0,C 180,E1 -10648.73,E2 -10648.73} C_VEL
LIN {X 0,Y 415.747,Z 380.483,A -85,B 0,C 180,E1 -10649.184,E2 -10649.184} C_VEL
LIN {X 0,Y 415.257,Z 392.681,A -85,B 0,C 180,E1 -10649.792,E2 -10649.792} C_VEL
LIN {X 0,Y 414.517,Z 404.274,A -85,B 0,C 180,E1 -10650.563,E2 -10650.563} C_VEL
LIN {X 0,Y 413.665,Z 416.606,A -85,B 0,C 180,E1 -10651.628,E2 -10651.628} C_VEL
LIN {X 0,Y 412.879,Z 426.512,A -85,B 0,C 180,E1 -10652.704,E2 -10652.704} C_VEL
LIN {X 0,Y 412.104,Z 436.233,A -85,B 0,C 180,E1 -10654.015,E2 -10654.015} C_VEL
LIN {X 0,Y 411.372,Z 445.122,A -85,B 0,C 180,E1 -10655.501,E2 -10655.501} C_VEL
LIN {X 0,Y 410.831,Z 452.573,A -85,B 0,C 180,E1 -10657.075,E2 -10657.075} C_VEL
LIN {X 0,Y 410.439,Z 458.504,A -85,B 0,C 180,E1 -10658.67,E2 -10658.67} C_VEL
LIN {X 0,Y 410.158,Z 462.542,A -85,B 0,C 180,E1 -10660.056,E2 -10660.056} C_VEL
LIN {X 0,Y 410.019,Z 464.852,A -85,B 0,C 180,E1 -10661.049,E2 -10661.049} C_VEL
LIN {X 0,Y 409.868,Z 467.395,A -85,B 0,C 180,E1 -10662.5,E2 -10662.5} C_VEL
LIN {X 0,Y 409.767,Z 468.997,A -85,B 0,C 180,E1 -10663.92,E2 -10663.92} C_VEL
LIN {X 0,Y 409.738,Z 469.752,A -85,B 0,C 180,E1 -10665.315,E2 -10665.315} C_VEL
LIN {X 0,Y 409.707,Z 469.713,A -85,B 0,C 180,E1 -10666.677,E2 -10666.677} C_VEL
LIN {X 0,Y 409.738,Z 468.88,A -85,B 0,C 180,E1 -10668.017,E2 -10668.017} C_VEL
LIN {X 0,Y 409.823,Z 467.336,A -85,B 0,C 180,E1 -10669.336,E2 -10669.336} C_VEL
LIN {X 0,Y 409.953,Z 465.096,A -85,B 0,C 180,E1 -10670.634,E2 -10670.634} C_VEL
LIN {X 0,Y 410.138,Z 461.853,A -85,B 0,C 180,E1 -10672.006,E2 -10672.006} C_VEL
LIN {X 0,Y 410.417,Z 456.973,A -85,B 0,C 180,E1 -10673.577,E2 -10673.577} C_VEL
LIN {X 0,Y 410.82,Z 450.5,A -85,B 0,C 180,E1 -10675.183,E2 -10675.183} C_VEL
LIN {X 0,Y 411.262,Z 443.582,A -85,B 0,C 180,E1 -10676.56,E2 -10676.56} C_VEL
LIN {X 0,Y 411.874,Z 435.171,A -85,B 0,C 180,E1 -10677.923,E2 -10677.923} C_VEL
LIN {X 0,Y 412.586,Z 424.813,A -85,B 0,C 180,E1 -10679.271,E2 -10679.271} C_VEL
LIN {X 0,Y 413.37,Z 413.288,A -85,B 0,C 180,E1 -10680.461,E2 -10680.461} C_VEL
LIN {X 0,Y 414.075,Z 401.402,A -85,B 0,C 180,E1 -10681.42,E2 -10681.42} C_VEL
LIN {X 0,Y 414.781,Z 389.372,A -85,B 0,C 180,E1 -10682.162,E2 -10682.162} C_VEL
LIN {X 0,Y 415.257,Z 376.598,A -85,B 0,C 180,E1 -10682.743,E2 -10682.743} C_VEL
LIN {X 0,Y 415.605,Z 364.099,A -85,B 0,C 180,E1 -10683.113,E2 -10683.113} C_VEL
LIN {X 0,Y 416.683,Z 280.106,A -85,B 0,C 180,E1 -10684.65,E2 -10684.65} C_VEL
LIN {X 0,Y 412.95,Z 259.401,A -85,B 0,C 180,E1 -10685.225,E2 -10685.225} C_VEL
LIN {X 0,Y 412.898,Z 258.328,A -85,B 0,C 180,E1 -10685.356,E2 -10685.356} C_VEL
LIN {X 0,Y 413.503,Z 248.925,A -85,B 0,C 180,E1 -10687.519,E2 -10687.519} C_VEL
LIN {X 0,Y 413.252,Z 246.492,A -85,B 0,C 180,E1 -10688.11,E2 -10688.11} C_VEL
LIN {X 0,Y 412.274,Z 244.732,A -85,B 0,C 180,E1 -10688.584,E2 -10688.584} C_VEL
LIN {X 0,Y 408.926,Z 242.416,A -85,B 0,C 180,E1 -10689.333,E2 -10689.333} C_VEL
LIN {X 0,Y 405.538,Z 240.125,A -85,B 0,C 180,E1 -10690.094,E2 -10690.094} C_VEL
LIN {X 0,Y 404.517,Z 238.393,A -85,B 0,C 180,E1 -10690.583,E2 -10690.583} C_VEL
LIN {X 0,Y 404.156,Z 236.672,A -85,B 0,C 180,E1 -10691.105,E2 -10691.105} C_VEL
LIN {X 0,Y 404.16,Z 236.64,A -85,B 0,C 180,E1 -10693.848,E2 -10693.848} C_VEL
LIN {X 0,Y 404.209,Z 236.633,A -85,B 0,C 180,E1 -10696.938,E2 -10696.938} C_VEL
LIN {X 0,Y 404.2,Z 236.632,A -85,B 0,C 180,E1 -10699.989,E2 -10699.989} C_VEL
LIN {X 0,Y 404.333,Z 236.619,A -85,B 0,C 180,E1 -10703.013,E2 -10703.013} C_VEL
LIN {X 0,Y 404.22,Z 236.634,A -85,B 0,C 180,E1 -10705.015,E2 -10705.015} C_VEL
LIN {X 0,Y 404.411,Z 236.605,A -85,B 0,C 180,E1 -10708.01,E2 -10708.01} C_VEL
LIN {X 0,Y 404.539,Z 236.589,A -85,B 0,C 180,E1 -10710.002,E2 -10710.002} C_VEL
LIN {X 0,Y 404.36,Z 236.618,A -85,B 0,C 180,E1 -10712.991,E2 -10712.991} C_VEL
LIN {X 0,Y 404.365,Z 236.611,A -85,B 0,C 180,E1 -10715.987,E2 -10715.987} C_VEL
LIN {X 0,Y 404.226,Z 236.632,A -85,B 0,C 180,E1 -10719.004,E2 -10719.004} C_VEL
LIN {X 0,Y 404.203,Z 236.632,A -85,B 0,C 180,E1 -10722.045,E2 -10722.045} C_VEL
LIN {X 0,Y 404.142,Z 236.642,A -85,B 0,C 180,E1 -10725.122,E2 -10725.122} C_VEL
LIN {X 0,Y 404.142,Z 236.64,A -85,B 0,C 180,E1 -10728.243,E2 -10728.243} C_VEL
LIN {X 0,Y 404.073,Z 236.651,A -85,B 0,C 180,E1 -10731.424,E2 -10731.424} C_VEL
LIN {X 0,Y 404.116,Z 236.642,A -85,B 0,C 180,E1 -10734.671,E2 -10734.671} C_VEL
LIN {X 0,Y 404.139,Z 236.646,A -85,B 0,C 180,E1 -10738.005,E2 -10738.005} C_VEL
LIN {X 0,Y 404.091,Z 236.647,A -85,B 0,C 180,E1 -10741.566,E2 -10741.566} C_VEL
LIN {X 0,Y 404.132,Z 236.64,A -85,B 0,C 180,E1 -10745.023,E2 -10745.023} C_VEL
LIN {X 0,Y 404.114,Z 236.645,A -85,B 0,C 180,E1 -10748.763,E2 -10748.763} C_VEL
LIN {X 0,Y 404.146,Z 236.638,A -85,B 0,C 180,E1 -10751.618,E2 -10751.618} C_VEL
LIN {X 0,Y 404.155,Z 236.645,A -85,B 0,C 180,E1 -10754.537,E2 -10754.537} C_VEL
LIN {X 0,Y 404.172,Z 236.636,A -85,B 0,C 180,E1 -10757.313,E2 -10757.313} C_VEL
LIN {X 0,Y 404.134,Z 236.64,A -85,B 0,C 180,E1 -10759.963,E2 -10759.963} C_VEL
LIN {X 0,Y 404.108,Z 236.647,A -85,B 0,C 180,E1 -10763.132,E2 -10763.132} C_VEL
LIN {X 0,Y 404.116,Z 236.642,A -85,B 0,C 180,E1 -10766.196,E2 -10766.196} C_VEL
LIN {X 0,Y 404.121,Z 236.642,A -85,B 0,C 180,E1 -10769.723,E2 -10769.723} C_VEL
LIN {X 0,Y 404.175,Z 236.642,A -85,B 0,C 180,E1 -10773.131,E2 -10773.131} C_VEL
LIN {X 0,Y 404.156,Z 236.643,A -85,B 0,C 180,E1 -10775.342,E2 -10775.342} C_VEL
LIN {X 0,Y 404.123,Z 236.641,A -85,B 0,C 180,E1 -10778.588,E2 -10778.588} C_VEL
LIN {X 0,Y 404.193,Z 236.636,A -85,B 0,C 180,E1 -10781.769,E2 -10781.769} C_VEL
LIN {X 0,Y 404.197,Z 236.633,A -85,B 0,C 180,E1 -10784.89,E2 -10784.89} C_VEL
LIN {X 0,Y 404.25,Z 236.629,A -85,B 0,C 180,E1 -10787.966,E2 -10787.966} C_VEL
LIN {X 0,Y 404.264,Z 236.624,A -85,B 0,C 180,E1 -10791.006,E2 -10791.006} C_VEL
LIN {X 0,Y 404.381,Z 236.614,A -85,B 0,C 180,E1 -10794.021,E2 -10794.021} C_VEL
LIN {X 0,Y 404.481,Z 236.604,A -85,B 0,C 180,E1 -10798.015,E2 -10798.015} C_VEL
LIN {X 0,Y 404.401,Z 236.606,A -85,B 0,C 180,E1 -10801.002,E2 -10801.002} C_VEL
LIN {X 0,Y 404.395,Z 236.607,A -85,B 0,C 180,E1 -10802.995,E2 -10802.995} C_VEL
LIN {X 0,Y 404.388,Z 236.612,A -85,B 0,C 180,E1 -10805.992,E2 -10805.992} C_VEL
LIN {X 0,Y 404.27,Z 236.624,A -85,B 0,C 180,E1 -10809.007,E2 -10809.007} C_VEL
LIN {X 0,Y 404.268,Z 236.626,A -85,B 0,C 180,E1 -10812.047,E2 -10812.047} C_VEL
LIN {X 0,Y 404.219,Z 236.631,A -85,B 0,C 180,E1 -10815.123,E2 -10815.123} C_VEL
LIN {X 0,Y 404.221,Z 236.631,A -85,B 0,C 180,E1 -10818.243,E2 -10818.243} C_VEL
LIN {X 0,Y 404.156,Z 236.638,A -85,B 0,C 180,E1 -10821.424,E2 -10821.424} C_VEL
LIN {X 0,Y 404.167,Z 236.64,A -85,B 0,C 180,E1 -10824.672,E2 -10824.672} C_VEL
LIN {X 0,Y 404.123,Z 236.641,A -85,B 0,C 180,E1 -10828.01,E2 -10828.01} C_VEL
LIN {X 0,Y 404.163,Z 236.636,A -85,B 0,C 180,E1 -10830.289,E2 -10830.289} C_VEL
LIN {X 0,Y 404.159,Z 236.638,A -85,B 0,C 180,E1 -10833.816,E2 -10833.816} C_VEL
LIN {X 0,Y 404.156,Z 236.639,A -85,B 0,C 180,E1 -10836.877,E2 -10836.877} C_VEL
LIN {X 0,Y 404.14,Z 236.64,A -85,B 0,C 180,E1 -10840.077,E2 -10840.077} C_VEL
LIN {X 0,Y 404.099,Z 236.646,A -85,B 0,C 180,E1 -10843.074,E2 -10843.074} C_VEL
LIN {X 0,Y 404.134,Z 236.644,A -85,B 0,C 180,E1 -10845.923,E2 -10845.923} C_VEL
LIN {X 0,Y 404.12,Z 236.641,A -85,B 0,C 180,E1 -10848.633,E2 -10848.633} C_VEL
LIN {X 0,Y 404.159,Z 236.64,A -85,B 0,C 180,E1 -10851.497,E2 -10851.497} C_VEL
LIN {X 0,Y 404.197,Z 236.632,A -85,B 0,C 180,E1 -10854.984,E2 -10854.984} C_VEL
LIN {X 0,Y 404.159,Z 236.643,A -85,B 0,C 180,E1 -10858.443,E2 -10858.443} C_VEL
LIN {X 0,Y 404.177,Z 236.64,A -85,B 0,C 180,E1 -10860.863,E2 -10860.863} C_VEL
LIN {X 0,Y 404.207,Z 236.703,A -85,B 0,C 180,E1 -10863.021,E2 -10863.021} C_VEL
LIN {X 0,Y 405.943,Z 245.424,A -85,B 0,C 180,E1 -10865.174,E2 -10865.174} C_VEL
LIN {X 0,Y 407.034,Z 251.51,A -85,B 0,C 180,E1 -10866.6,E2 -10866.6} C_VEL
LIN {X 0,Y 406.063,Z 265.924,A -85,B 0,C 180,E1 -10869.746,E2 -10869.746} C_VEL
LIN {X 0,Y 405.84,Z 269.479,A -85,B 0,C 180,E1 -10870.46,E2 -10870.46} C_VEL
LIN {X 0,Y 406.72,Z 275.292,A -85,B 0,C 180,E1 -10870.654,E2 -10870.654} C_VEL
LIN {X 0,Y 409.928,Z 295.522,A -85,B 0,C 180,E1 -10871.181,E2 -10871.181} C_VEL
LIN {X 0,Y 408.74,Z 377.203,A -85,B 0,C 180,E1 -10872.713,E2 -10872.713} C_VEL
LIN {X 0,Y 408.254,Z 391.023,A -85,B 0,C 180,E1 -10873.175,E2 -10873.175} C_VEL
LIN {X 0,Y 407.654,Z 403.504,A -85,B 0,C 180,E1 -10873.794,E2 -10873.794} C_VEL
LIN {X 0,Y 406.857,Z 415.456,A -85,B 0,C 180,E1 -10874.597,E2 -10874.597} C_VEL
LIN {X 0,Y 406.093,Z 426.946,A -85,B 0,C 180,E1 -10875.594,E2 -10875.594} C_VEL
LIN {X 0,Y 405.354,Z 437.304,A -85,B 0,C 180,E1 -10876.717,E2 -10876.717} C_VEL
LIN {X 0,Y 404.675,Z 446.599,A -85,B 0,C 180,E1 -10877.97,E2 -10877.97} C_VEL
LIN {X 0,Y 404.001,Z 455.631,A -85,B 0,C 180,E1 -10879.474,E2 -10879.474} C_VEL
LIN {X 0,Y 403.557,Z 462.894,A -85,B 0,C 180,E1 -10880.981,E2 -10880.981} C_VEL
LIN {X 0,Y 403.177,Z 468.671,A -85,B 0,C 180,E1 -10882.486,E2 -10882.486} C_VEL
LIN {X 0,Y 402.985,Z 473.21,A -85,B 0,C 180,E1 -10883.992,E2 -10883.992} C_VEL
LIN {X 0,Y 402.949,Z 475.599,A -85,B 0,C 180,E1 -10884.995,E2 -10884.995} C_VEL
LIN {X 0,Y 402.849,Z 477.55,A -85,B 0,C 180,E1 -10885.997,E2 -10885.997} C_VEL
LIN {X 0,Y 402.791,Z 479.07,A -85,B 0,C 180,E1 -10886.998,E2 -10886.998} C_VEL
LIN {X 0,Y 402.83,Z 480.132,A -85,B 0,C 180,E1 -10887.999,E2 -10887.999} C_VEL
LIN {X 0,Y 402.853,Z 480.796,A -85,B 0,C 180,E1 -10888.999,E2 -10888.999} C_VEL
LIN {X 0,Y 402.84,Z 481.067,A -85,B 0,C 180,E1 -10889.998,E2 -10889.998} C_VEL
LIN {X 0,Y 402.853,Z 480.931,A -85,B 0,C 180,E1 -10890.998,E2 -10890.998} C_VEL
LIN {X 0,Y 402.829,Z 480.357,A -85,B 0,C 180,E1 -10891.998,E2 -10891.998} C_VEL
LIN {X 0,Y 402.851,Z 478.021,A -85,B 0,C 180,E1 -10894,E2 -10894} C_VEL
LIN {X 0,Y 402.979,Z 475.127,A -85,B 0,C 180,E1 -10895.503,E2 -10895.503} C_VEL
LIN {X 0,Y 403.117,Z 471.193,A -85,B 0,C 180,E1 -10897.008,E2 -10897.008} C_VEL
LIN {X 0,Y 403.458,Z 466.117,A -85,B 0,C 180,E1 -10898.513,E2 -10898.513} C_VEL
LIN {X 0,Y 403.89,Z 459.744,A -85,B 0,C 180,E1 -10900.019,E2 -10900.019} C_VEL
LIN {X 0,Y 404.523,Z 451.771,A -85,B 0,C 180,E1 -10901.523,E2 -10901.523} C_VEL
LIN {X 0,Y 405.468,Z 441.861,A -85,B 0,C 180,E1 -10903.02,E2 -10903.02} C_VEL
LIN {X 0,Y 406.184,Z 432.226,A -85,B 0,C 180,E1 -10904.194,E2 -10904.194} C_VEL
LIN {X 0,Y 406.985,Z 421.284,A -85,B 0,C 180,E1 -10905.267,E2 -10905.267} C_VEL
LIN {X 0,Y 407.824,Z 410.137,A -85,B 0,C 180,E1 -10906.132,E2 -10906.132} C_VEL
LIN {X 0,Y 408.588,Z 398.912,A -85,B 0,C 180,E1 -10906.807,E2 -10906.807} C_VEL
LIN {X 0,Y 409.15,Z 386.421,A -85,B 0,C 180,E1 -10907.363,E2 -10907.363} C_VEL
LIN {X 0,Y 409.588,Z 373.64,A -85,B 0,C 180,E1 -10907.73,E2 -10907.73} C_VEL
LIN {X 0,Y 410.814,Z 295.016,A -85,B 0,C 180,E1 -10909.22,E2 -10909.22} C_VEL
LIN {X 0,Y 407.021,Z 272.864,A -85,B 0,C 180,E1 -10909.88,E2 -10909.88} C_VEL
LIN {X 0,Y 406.205,Z 268.683,A -85,B 0,C 180,E1 -10910.043,E2 -10910.043} C_VEL
LIN {X 0,Y 407.251,Z 252.786,A -85,B 0,C 180,E1 -10913.383,E2 -10913.383} C_VEL
LIN {X 0,Y 405.699,Z 243.699,A -85,B 0,C 180,E1 -10915.493,E2 -10915.493} C_VEL
LIN {X 0,Y 404.234,Z 236.716,A -85,B 0,C 180,E1 -10917.233,E2 -10917.233} C_VEL
LIN {X 0,Y 404.155,Z 236.64,A -85,B 0,C 180,E1 -10920.282,E2 -10920.282} C_VEL
LIN {X 0,Y 404.154,Z 236.644,A -85,B 0,C 180,E1 -10923.809,E2 -10923.809} C_VEL
LIN {X 0,Y 404.142,Z 236.642,A -85,B 0,C 180,E1 -10926.87,E2 -10926.87} C_VEL
LIN {X 0,Y 404.125,Z 236.648,A -85,B 0,C 180,E1 -10930.071,E2 -10930.071} C_VEL
LIN {X 0,Y 404.148,Z 236.638,A -85,B 0,C 180,E1 -10933.078,E2 -10933.078} C_VEL
LIN {X 0,Y 404.125,Z 236.644,A -85,B 0,C 180,E1 -10935.918,E2 -10935.918} C_VEL
LIN {X 0,Y 404.106,Z 236.649,A -85,B 0,C 180,E1 -10938.628,E2 -10938.628} C_VEL
LIN {X 0,Y 404.14,Z 236.64,A -85,B 0,C 180,E1 -10941.491,E2 -10941.491} C_VEL
LIN {X 0,Y 404.174,Z 236.639,A -85,B 0,C 180,E1 -10944.978,E2 -10944.978} C_VEL
LIN {X 0,Y 404.139,Z 236.646,A -85,B 0,C 180,E1 -10948.438,E2 -10948.438} C_VEL
LIN {X 0,Y 404.149,Z 236.642,A -85,B 0,C 180,E1 -10950.857,E2 -10950.857} C_VEL
LIN {X 0,Y 404.151,Z 236.642,A -85,B 0,C 180,E1 -10954.718,E2 -10954.718} C_VEL
LIN {X 0,Y 404.16,Z 236.635,A -85,B 0,C 180,E1 -10957.502,E2 -10957.502} C_VEL
LIN {X 0,Y 404.129,Z 236.642,A -85,B 0,C 180,E1 -10960.7,E2 -10960.7} C_VEL
LIN {X 0,Y 404.171,Z 236.634,A -85,B 0,C 180,E1 -10963.84,E2 -10963.84} C_VEL
LIN {X 0,Y 404.275,Z 236.626,A -85,B 0,C 180,E1 -10966.933,E2 -10966.933} C_VEL
LIN {X 0,Y 404.237,Z 236.629,A -85,B 0,C 180,E1 -10969.982,E2 -10969.982} C_VEL
LIN {X 0,Y 404.368,Z 236.618,A -85,B 0,C 180,E1 -10973.006,E2 -10973.006} C_VEL
LIN {X 0,Y 404.251,Z 236.628,A -85,B 0,C 180,E1 -10975.007,E2 -10975.007} C_VEL
LIN {X 0,Y 404.456,Z 236.602,A -85,B 0,C 180,E1 -10978.002,E2 -10978.002} C_VEL
LIN {X 0,Y 404.588,Z 236.583,A -85,B 0,C 180,E1 -10979.993,E2 -10979.993} C_VEL
LIN {X 0,Y 404.395,Z 236.61,A -85,B 0,C 180,E1 -10982.982,E2 -10982.982} C_VEL
LIN {X 0,Y 404.357,Z 236.616,A -85,B 0,C 180,E1 -10986.981,E2 -10986.981} C_VEL
LIN {X 0,Y 404.246,Z 236.63,A -85,B 0,C 180,E1 -10990.005,E2 -10990.005} C_VEL
LIN {X 0,Y 404.238,Z 236.633,A -85,B 0,C 180,E1 -10993.205,E2 -10993.205} C_VEL
LIN {X 0,Y 404.184,Z 236.639,A -85,B 0,C 180,E1 -10997,E2 -10997} C_VEL
LIN {X 0,Y 404.198,Z 236.636,A -85,B 0,C 180,E1 -11000.873,E2 -11000.873} C_VEL
LIN {X 0,Y 404.212,Z 236.889,A -85,B 0,C 180,E1 -11001.273,E2 -11001.273} C_VEL
LIN {X 0,Y 406.697,Z 248.376,A -85,B 0,C 180,E1 -11003.95,E2 -11003.95} C_VEL
LIN {X 0,Y 406.68,Z 252.241,A -85,B 0,C 180,E1 -11004.767,E2 -11004.767} C_VEL
LIN {X 0,Y 406.408,Z 258.603,A -85,B 0,C 180,E1 -11006.032,E2 -11006.032} C_VEL
LIN {X 0,Y 410.534,Z 278.941,A -85,B 0,C 180,E1 -11006.695,E2 -11006.695} C_VEL
LIN {X 0,Y 410.991,Z 283.824,A -85,B 0,C 180,E1 -11006.817,E2 -11006.817} C_VEL
LIN {X 0,Y 409.538,Z 367.143,A -85,B 0,C 180,E1 -11008.411,E2 -11008.411} C_VEL
LIN {X 0,Y 408.993,Z 380.915,A -85,B 0,C 180,E1 -11008.885,E2 -11008.885} C_VEL
LIN {X 0,Y 408.463,Z 393.485,A -85,B 0,C 180,E1 -11009.532,E2 -11009.532} C_VEL
LIN {X 0,Y 407.639,Z 405.379,A -85,B 0,C 180,E1 -11010.351,E2 -11010.351} C_VEL
LIN {X 0,Y 406.808,Z 416.627,A -85,B 0,C 180,E1 -11011.345,E2 -11011.345} C_VEL
LIN {X 0,Y 406.01,Z 426.58,A -85,B 0,C 180,E1 -11012.443,E2 -11012.443} C_VEL
LIN {X 0,Y 405.256,Z 435.776,A -85,B 0,C 180,E1 -11013.697,E2 -11013.697} C_VEL
LIN {X 0,Y 404.42,Z 444.944,A -85,B 0,C 180,E1 -11015.242,E2 -11015.242} C_VEL
LIN {X 0,Y 403.844,Z 452.38,A -85,B 0,C 180,E1 -11016.824,E2 -11016.824} C_VEL
LIN {X 0,Y 403.403,Z 458.147,A -85,B 0,C 180,E1 -11018.377,E2 -11018.377} C_VEL
LIN {X 0,Y 403.063,Z 463.228,A -85,B 0,C 180,E1 -11020.165,E2 -11020.165} C_VEL
LIN {X 0,Y 402.847,Z 466.048,A -85,B 0,C 180,E1 -11021.512,E2 -11021.512} C_VEL
LIN {X 0,Y 402.753,Z 468.107,A -85,B 0,C 180,E1 -11022.874,E2 -11022.874} C_VEL
LIN {X 0,Y 402.652,Z 469.447,A -85,B 0,C 180,E1 -11024.309,E2 -11024.309} C_VEL
LIN {X 0,Y 402.632,Z 469.919,A -85,B 0,C 180,E1 -11025.72,E2 -11025.72} C_VEL
LIN {X 0,Y 402.611,Z 469.59,A -85,B 0,C 180,E1 -11027.138,E2 -11027.138} C_VEL
LIN {X 0,Y 402.678,Z 468.387,A -85,B 0,C 180,E1 -11028.618,E2 -11028.618} C_VEL
LIN {X 0,Y 402.782,Z 466.209,A -85,B 0,C 180,E1 -11030.136,E2 -11030.136} C_VEL
LIN {X 0,Y 403.01,Z 462.956,A -85,B 0,C 180,E1 -11031.681,E2 -11031.681} C_VEL
LIN {X 0,Y 403.29,Z 458.426,A -85,B 0,C 180,E1 -11033.269,E2 -11033.269} C_VEL
LIN {X 0,Y 403.645,Z 452.258,A -85,B 0,C 180,E1 -11034.933,E2 -11034.933} C_VEL
LIN {X 0,Y 404.177,Z 444.506,A -85,B 0,C 180,E1 -11036.561,E2 -11036.561} C_VEL
LIN {X 0,Y 404.895,Z 435.289,A -85,B 0,C 180,E1 -11038.095,E2 -11038.095} C_VEL
LIN {X 0,Y 405.602,Z 425.449,A -85,B 0,C 180,E1 -11039.406,E2 -11039.406} C_VEL
LIN {X 0,Y 406.379,Z 414.064,A -85,B 0,C 180,E1 -11040.614,E2 -11040.614} C_VEL
LIN {X 0,Y 407.112,Z 402.721,A -85,B 0,C 180,E1 -11041.567,E2 -11041.567} C_VEL
LIN {X 0,Y 407.84,Z 390.62,A -85,B 0,C 180,E1 -11042.344,E2 -11042.344} C_VEL
LIN {X 0,Y 408.383,Z 377.296,A -85,B 0,C 180,E1 -11042.974,E2 -11042.974} C_VEL
LIN {X 0,Y 408.756,Z 364.579,A -85,B 0,C 180,E1 -11043.367,E2 -11043.367} C_VEL
LIN {X 0,Y 409.902,Z 280.939,A -85,B 0,C 180,E1 -11044.926,E2 -11044.926} C_VEL
LIN {X 0,Y 406.018,Z 259.544,A -85,B 0,C 180,E1 -11045.531,E2 -11045.531} C_VEL
LIN {X 0,Y 405.971,Z 258.748,A -85,B 0,C 180,E1 -11045.603,E2 -11045.603} C_VEL
LIN {X 0,Y 406.551,Z 249.945,A -85,B 0,C 180,E1 -11047.649,E2 -11047.649} C_VEL
LIN {X 0,Y 405.155,Z 241.815,A -85,B 0,C 180,E1 -11049.703,E2 -11049.703} C_VEL
LIN {X 0,Y 404.517,Z 238.393,A -85,B 0,C 180,E1 -11050.583,E2 -11050.583} C_VEL
LIN {X 0,Y 403.908,Z 237.162,A -85,B 0,C 180,E1 -11051.085,E2 -11051.085} C_VEL
LIN {X 0,Y 402.341,Z 236.868,A -85,B 0,C 180,E1 -11051.881,E2 -11051.881} C_VEL
LIN {X 0,Y 398.153,Z 237.465,A -85,B 0,C 180,E1 -11053.809,E2 -11053.809} C_VEL
LIN {X 0,Y 397.187,Z 237.518,A -85,B 0,C 180,E1 -11054.677,E2 -11054.677} C_VEL
LIN {X 0,Y 397.107,Z 237.518,A -85,B 0,C 180,E1 -11054.97,E2 -11054.97} C_VEL
LIN {X 0,Y 397.158,Z 237.509,A -85,B 0,C 180,E1 -11057.742,E2 -11057.742} C_VEL
LIN {X 0,Y 397.185,Z 237.511,A -85,B 0,C 180,E1 -11060.838,E2 -11060.838} C_VEL
LIN {X 0,Y 397.312,Z 237.489,A -85,B 0,C 180,E1 -11063.909,E2 -11063.909} C_VEL
LIN {X 0,Y 397.38,Z 237.481,A -85,B 0,C 180,E1 -11067.975,E2 -11067.975} C_VEL
LIN {X 0,Y 397.509,Z 237.465,A -85,B 0,C 180,E1 -11070.002,E2 -11070.002} C_VEL
LIN {X 0,Y 397.319,Z 237.496,A -85,B 0,C 180,E1 -11073.044,E2 -11073.044} C_VEL
LIN {X 0,Y 397.314,Z 237.489,A -85,B 0,C 180,E1 -11076.094,E2 -11076.094} C_VEL
LIN {X 0,Y 397.188,Z 237.511,A -85,B 0,C 180,E1 -11079.165,E2 -11079.165} C_VEL
LIN {X 0,Y 397.162,Z 237.508,A -85,B 0,C 180,E1 -11082.261,E2 -11082.261} C_VEL
LIN {X 0,Y 397.114,Z 237.52,A -85,B 0,C 180,E1 -11085.396,E2 -11085.396} C_VEL
LIN {X 0,Y 397.095,Z 237.516,A -85,B 0,C 180,E1 -11088.578,E2 -11088.578} C_VEL
LIN {X 0,Y 397.032,Z 237.531,A -85,B 0,C 180,E1 -11091.824,E2 -11091.824} C_VEL
LIN {X 0,Y 397.096,Z 237.517,A -85,B 0,C 180,E1 -11095.137,E2 -11095.137} C_VEL
LIN {X 0,Y 397.105,Z 237.521,A -85,B 0,C 180,E1 -11097.782,E2 -11097.782} C_VEL
LIN {X 0,Y 397.031,Z 237.525,A -85,B 0,C 180,E1 -11100.888,E2 -11100.888} C_VEL
LIN {X 0,Y 397.073,Z 237.523,A -85,B 0,C 180,E1 -11104.5,E2 -11104.5} C_VEL
LIN {X 0,Y 397.06,Z 237.528,A -85,B 0,C 180,E1 -11108.281,E2 -11108.281} C_VEL
LIN {X 0,Y 397.111,Z 237.517,A -85,B 0,C 180,E1 -11112,E2 -11112} C_VEL
LIN {X 0,Y 397.11,Z 237.516,A -85,B 0,C 180,E1 -11115.067,E2 -11115.067} C_VEL
LIN {X 0,Y 397.119,Z 237.515,A -85,B 0,C 180,E1 -11118.014,E2 -11118.014} C_VEL
LIN {X 0,Y 397.076,Z 237.519,A -85,B 0,C 180,E1 -11121.734,E2 -11121.734} C_VEL
LIN {X 0,Y 397.096,Z 237.517,A -85,B 0,C 180,E1 -11125.515,E2 -11125.515} C_VEL
LIN {X 0,Y 397.053,Z 237.528,A -85,B 0,C 180,E1 -11129.126,E2 -11129.126} C_VEL
LIN {X 0,Y 397.173,Z 237.509,A -85,B 0,C 180,E1 -11132.618,E2 -11132.618} C_VEL
LIN {X 0,Y 397.111,Z 237.515,A -85,B 0,C 180,E1 -11135.989,E2 -11135.989} C_VEL
LIN {X 0,Y 397.126,Z 237.516,A -85,B 0,C 180,E1 -11139.713,E2 -11139.713} C_VEL
LIN {X 0,Y 397.172,Z 237.508,A -85,B 0,C 180,E1 -11142.853,E2 -11142.853} C_VEL
LIN {X 0,Y 397.224,Z 237.5,A -85,B 0,C 180,E1 -11146.71,E2 -11146.71} C_VEL
LIN {X 0,Y 397.213,Z 237.508,A -85,B 0,C 180,E1 -11149.816,E2 -11149.816} C_VEL
LIN {X 0,Y 397.295,Z 237.492,A -85,B 0,C 180,E1 -11152.894,E2 -11152.894} C_VEL
LIN {X 0,Y 397.24,Z 237.498,A -85,B 0,C 180,E1 -11154.932,E2 -11154.932} C_VEL
LIN {X 0,Y 397.45,Z 237.48,A -85,B 0,C 180,E1 -11157.98,E2 -11157.98} C_VEL
LIN {X 0,Y 397.446,Z 237.479,A -85,B 0,C 180,E1 -11162.033,E2 -11162.033} C_VEL
LIN {X 0,Y 397.339,Z 237.492,A -85,B 0,C 180,E1 -11166.098,E2 -11166.098} C_VEL
LIN {X 0,Y 397.241,Z 237.499,A -85,B 0,C 180,E1 -11169.168,E2 -11169.168} C_VEL
LIN {X 0,Y 397.232,Z 237.504,A -85,B 0,C 180,E1 -11172.264,E2 -11172.264} C_VEL
LIN {X 0,Y 397.193,Z 237.504,A -85,B 0,C 180,E1 -11175.397,E2 -11175.397} C_VEL
LIN {X 0,Y 397.175,Z 237.513,A -85,B 0,C 180,E1 -11178.578,E2 -11178.578} C_VEL
LIN {X 0,Y 397.113,Z 237.514,A -85,B 0,C 180,E1 -11181.823,E2 -11181.823} C_VEL
LIN {X 0,Y 397.116,Z 237.519,A -85,B 0,C 180,E1 -11185.14,E2 -11185.14} C_VEL
LIN {X 0,Y 397.083,Z 237.52,A -85,B 0,C 180,E1 -11188.552,E2 -11188.552} C_VEL
LIN {X 0,Y 397.101,Z 237.516,A -85,B 0,C 180,E1 -11191.839,E2 -11191.839} C_VEL
LIN {X 0,Y 397.141,Z 237.511,A -85,B 0,C 180,E1 -11194.497,E2 -11194.497} C_VEL
LIN {X 0,Y 397.114,Z 237.514,A -85,B 0,C 180,E1 -11198.279,E2 -11198.279} C_VEL
LIN {X 0,Y 397.067,Z 237.522,A -85,B 0,C 180,E1 -11200.917,E2 -11200.917} C_VEL
LIN {X 0,Y 397.097,Z 237.517,A -85,B 0,C 180,E1 -11204.931,E2 -11204.931} C_VEL
LIN {X 0,Y 397.06,Z 237.524,A -85,B 0,C 180,E1 -11208.028,E2 -11208.028} C_VEL
LIN {X 0,Y 397.113,Z 237.515,A -85,B 0,C 180,E1 -11211.147,E2 -11211.147} C_VEL
LIN {X 0,Y 397.122,Z 237.514,A -85,B 0,C 180,E1 -11214.502,E2 -11214.502} C_VEL
LIN {X 0,Y 397.135,Z 237.512,A -85,B 0,C 180,E1 -11216.728,E2 -11216.728} C_VEL
LIN {X 0,Y 397.139,Z 237.518,A -85,B 0,C 180,E1 -11220.296,E2 -11220.296} C_VEL
LIN {X 0,Y 397.15,Z 237.669,A -85,B 0,C 180,E1 -11222.819,E2 -11222.819} C_VEL
LIN {X 0,Y 399.376,Z 248.832,A -85,B 0,C 180,E1 -11225.572,E2 -11225.572} C_VEL
LIN {X 0,Y 400.09,Z 253.683,A -85,B 0,C 180,E1 -11226.718,E2 -11226.718} C_VEL
LIN {X 0,Y 398.919,Z 269.119,A -85,B 0,C 180,E1 -11230.107,E2 -11230.107} C_VEL
LIN {X 0,Y 399.266,Z 271.89,A -85,B 0,C 180,E1 -11230.252,E2 -11230.252} C_VEL
LIN {X 0,Y 403.136,Z 296.12,A -85,B 0,C 180,E1 -11230.9,E2 -11230.9} C_VEL
LIN {X 0,Y 401.914,Z 377.063,A -85,B 0,C 180,E1 -11232.442,E2 -11232.442} C_VEL
LIN {X 0,Y 401.41,Z 390.887,A -85,B 0,C 180,E1 -11232.912,E2 -11232.912} C_VEL
LIN {X 0,Y 400.811,Z 402.821,A -85,B 0,C 180,E1 -11233.509,E2 -11233.509} C_VEL
LIN {X 0,Y 399.962,Z 414.944,A -85,B 0,C 180,E1 -11234.324,E2 -11234.324} C_VEL
LIN {X 0,Y 399.146,Z 427.015,A -85,B 0,C 180,E1 -11235.388,E2 -11235.388} C_VEL
LIN {X 0,Y 398.413,Z 437.142,A -85,B 0,C 180,E1 -11236.507,E2 -11236.507} C_VEL
LIN {X 0,Y 397.701,Z 446.293,A -85,B 0,C 180,E1 -11237.755,E2 -11237.755} C_VEL
LIN {X 0,Y 396.98,Z 455.363,A -85,B 0,C 180,E1 -11239.285,E2 -11239.285} C_VEL
LIN {X 0,Y 396.511,Z 462.663,A -85,B 0,C 180,E1 -11240.819,E2 -11240.819} C_VEL
LIN {X 0,Y 396.11,Z 468.475,A -85,B 0,C 180,E1 -11242.351,E2 -11242.351} C_VEL
LIN {X 0,Y 395.869,Z 473.717,A -85,B 0,C 180,E1 -11244.159,E2 -11244.159} C_VEL
LIN {X 0,Y 395.774,Z 477.402,A -85,B 0,C 180,E1 -11245.925,E2 -11245.925} C_VEL
LIN {X 0,Y 395.698,Z 478.938,A -85,B 0,C 180,E1 -11246.944,E2 -11246.944} C_VEL
LIN {X 0,Y 395.727,Z 480.012,A -85,B 0,C 180,E1 -11247.963,E2 -11247.963} C_VEL
LIN {X 0,Y 395.765,Z 480.685,A -85,B 0,C 180,E1 -11248.981,E2 -11248.981} C_VEL
LIN {X 0,Y 395.768,Z 480.964,A -85,B 0,C 180,E1 -11249.998,E2 -11249.998} C_VEL
LIN {X 0,Y 395.764,Z 480.841,A -85,B 0,C 180,E1 -11251.016,E2 -11251.016} C_VEL
LIN {X 0,Y 395.726,Z 480.277,A -85,B 0,C 180,E1 -11252.034,E2 -11252.034} C_VEL
LIN {X 0,Y 395.778,Z 477.955,A -85,B 0,C 180,E1 -11254.071,E2 -11254.071} C_VEL
LIN {X 0,Y 395.882,Z 474.524,A -85,B 0,C 180,E1 -11255.855,E2 -11255.855} C_VEL
LIN {X 0,Y 396.169,Z 469.608,A -85,B 0,C 180,E1 -11257.644,E2 -11257.644} C_VEL
LIN {X 0,Y 396.639,Z 463.118,A -85,B 0,C 180,E1 -11259.431,E2 -11259.431} C_VEL
LIN {X 0,Y 397.186,Z 456.022,A -85,B 0,C 180,E1 -11260.963,E2 -11260.963} C_VEL
LIN {X 0,Y 398.047,Z 447.157,A -85,B 0,C 180,E1 -11262.489,E2 -11262.489} C_VEL
LIN {X 0,Y 398.951,Z 437.094,A -85,B 0,C 180,E1 -11263.886,E2 -11263.886} C_VEL
LIN {X 0,Y 399.687,Z 426.824,A -85,B 0,C 180,E1 -11265.03,E2 -11265.03} C_VEL
LIN {X 0,Y 400.646,Z 415.461,A -85,B 0,C 180,E1 -11266.036,E2 -11266.036} C_VEL
LIN {X 0,Y 401.473,Z 403.698,A -85,B 0,C 180,E1 -11266.852,E2 -11266.852} C_VEL
LIN {X 0,Y 402.268,Z 391.57,A -85,B 0,C 180,E1 -11267.472,E2 -11267.472} C_VEL
LIN {X 0,Y 402.734,Z 378.384,A -85,B 0,C 180,E1 -11267.944,E2 -11267.944} C_VEL
LIN {X 0,Y 403.339,Z 352.249,A -85,B 0,C 180,E1 -11268.472,E2 -11268.472} C_VEL
LIN {X 0,Y 404.15,Z 295.665,A -85,B 0,C 180,E1 -11269.575,E2 -11269.575} C_VEL
LIN {X 0,Y 400.422,Z 273.823,A -85,B 0,C 180,E1 -11270.246,E2 -11270.246} C_VEL
LIN {X 0,Y 399.379,Z 268.55,A -85,B 0,C 180,E1 -11270.45,E2 -11270.45} C_VEL
LIN {X 0,Y 400.342,Z 254.128,A -85,B 0,C 180,E1 -11273.537,E2 -11273.537} C_VEL
LIN {X 0,Y 398.985,Z 246.029,A -85,B 0,C 180,E1 -11275.451,E2 -11275.451} C_VEL
LIN {X 0,Y 397.213,Z 237.705,A -85,B 0,C 180,E1 -11277.527,E2 -11277.527} C_VEL
LIN {X 0,Y 397.088,Z 237.519,A -85,B 0,C 180,E1 -11280.879,E2 -11280.879} C_VEL
LIN {X 0,Y 397.134,Z 237.516,A -85,B 0,C 180,E1 -11284.49,E2 -11284.49} C_VEL
LIN {X 0,Y 397.099,Z 237.523,A -85,B 0,C 180,E1 -11288.273,E2 -11288.273} C_VEL
LIN {X 0,Y 397.058,Z 237.527,A -85,B 0,C 180,E1 -11291.972,E2 -11291.972} C_VEL
LIN {X 0,Y 397.09,Z 237.518,A -85,B 0,C 180,E1 -11295.065,E2 -11295.065} C_VEL
LIN {X 0,Y 397.056,Z 237.525,A -85,B 0,C 180,E1 -11298.019,E2 -11298.019} C_VEL
LIN {X 0,Y 397.092,Z 237.519,A -85,B 0,C 180,E1 -11301.718,E2 -11301.718} C_VEL
LIN {X 0,Y 397.118,Z 237.516,A -85,B 0,C 180,E1 -11305.501,E2 -11305.501} C_VEL
LIN {X 0,Y 397.076,Z 237.52,A -85,B 0,C 180,E1 -11309.112,E2 -11309.112} C_VEL
LIN {X 0,Y 397.061,Z 237.526,A -85,B 0,C 180,E1 -11312.247,E2 -11312.247} C_VEL
LIN {X 0,Y 397.1,Z 237.522,A -85,B 0,C 180,E1 -11314.859,E2 -11314.859} C_VEL
LIN {X 0,Y 397.086,Z 237.518,A -85,B 0,C 180,E1 -11318.175,E2 -11318.175} C_VEL
LIN {X 0,Y 397.082,Z 237.52,A -85,B 0,C 180,E1 -11321.417,E2 -11321.417} C_VEL
LIN {X 0,Y 397.114,Z 237.514,A -85,B 0,C 180,E1 -11324.6,E2 -11324.6} C_VEL
LIN {X 0,Y 397.208,Z 237.5,A -85,B 0,C 180,E1 -11327.736,E2 -11327.736} C_VEL
LIN {X 0,Y 397.218,Z 237.504,A -85,B 0,C 180,E1 -11330.831,E2 -11330.831} C_VEL
LIN {X 0,Y 397.333,Z 237.486,A -85,B 0,C 180,E1 -11333.902,E2 -11333.902} C_VEL
LIN {X 0,Y 397.425,Z 237.478,A -85,B 0,C 180,E1 -11337.967,E2 -11337.967} C_VEL
LIN {X 0,Y 397.558,Z 237.459,A -85,B 0,C 180,E1 -11339.993,E2 -11339.993} C_VEL
LIN {X 0,Y 397.354,Z 237.487,A -85,B 0,C 180,E1 -11343.035,E2 -11343.035} C_VEL
LIN {X 0,Y 397.309,Z 237.494,A -85,B 0,C 180,E1 -11347.106,E2 -11347.106} C_VEL
LIN {X 0,Y 397.203,Z 237.506,A -85,B 0,C 180,E1 -11350.184,E2 -11350.184} C_VEL
LIN {X 0,Y 397.198,Z 237.511,A -85,B 0,C 180,E1 -11353.314,E2 -11353.314} C_VEL
LIN {X 0,Y 397.15,Z 237.514,A -85,B 0,C 180,E1 -11357.148,E2 -11357.148} C_VEL
LIN {X 0,Y 397.179,Z 237.614,A -85,B 0,C 180,E1 -11360.853,E2 -11360.853} C_VEL
LIN {X 0,Y 399.704,Z 249.302,A -85,B 0,C 180,E1 -11363.672,E2 -11363.672} C_VEL
LIN {X 0,Y 399.9,Z 252.528,A -85,B 0,C 180,E1 -11364.384,E2 -11364.384} C_VEL
LIN {X 0,Y 399.588,Z 258.612,A -85,B 0,C 180,E1 -11365.621,E2 -11365.621} C_VEL
LIN {X 0,Y 403.992,Z 280.231,A -85,B 0,C 180,E1 -11366.35,E2 -11366.35} C_VEL
LIN {X 0,Y 404.392,Z 284.285,A -85,B 0,C 180,E1 -11366.457,E2 -11366.457} C_VEL
LIN {X 0,Y 402.89,Z 366.592,A -85,B 0,C 180,E1 -11368.063,E2 -11368.063} C_VEL
LIN {X 0,Y 402.355,Z 380.315,A -85,B 0,C 180,E1 -11368.535,E2 -11368.535} C_VEL
LIN {X 0,Y 401.814,Z 391.929,A -85,B 0,C 180,E1 -11369.123,E2 -11369.123} C_VEL
LIN {X 0,Y 401.04,Z 403.32,A -85,B 0,C 180,E1 -11369.881,E2 -11369.881} C_VEL
LIN {X 0,Y 400.132,Z 415.104,A -85,B 0,C 180,E1 -11370.903,E2 -11370.903} C_VEL
LIN {X 0,Y 399.189,Z 425.848,A -85,B 0,C 180,E1 -11372.075,E2 -11372.075} C_VEL
LIN {X 0,Y 398.362,Z 435.67,A -85,B 0,C 180,E1 -11373.419,E2 -11373.419} C_VEL
LIN {X 0,Y 397.455,Z 444.823,A -85,B 0,C 180,E1 -11374.979,E2 -11374.979} C_VEL
LIN {X 0,Y 396.917,Z 451.392,A -85,B 0,C 180,E1 -11376.371,E2 -11376.371} C_VEL
LIN {X 0,Y 396.416,Z 457.658,A -85,B 0,C 180,E1 -11378.025,E2 -11378.025} C_VEL
LIN {X 0,Y 396.039,Z 462.503,A -85,B 0,C 180,E1 -11379.694,E2 -11379.694} C_VEL
LIN {X 0,Y 395.833,Z 465.53,A -85,B 0,C 180,E1 -11381.054,E2 -11381.054} C_VEL
LIN {X 0,Y 395.685,Z 467.758,A -85,B 0,C 180,E1 -11382.437,E2 -11382.437} C_VEL
LIN {X 0,Y 395.582,Z 469.237,A -85,B 0,C 180,E1 -11383.846,E2 -11383.846} C_VEL
LIN {X 0,Y 395.536,Z 469.957,A -85,B 0,C 180,E1 -11385.281,E2 -11385.281} C_VEL
LIN {X 0,Y 395.504,Z 469.873,A -85,B 0,C 180,E1 -11386.752,E2 -11386.752} C_VEL
LIN {X 0,Y 395.548,Z 468.901,A -85,B 0,C 180,E1 -11388.252,E2 -11388.252} C_VEL
LIN {X 0,Y 395.695,Z 466.175,A -85,B 0,C 180,E1 -11390.256,E2 -11390.256} C_VEL
LIN {X 0,Y 395.905,Z 463.453,A -85,B 0,C 180,E1 -11391.591,E2 -11391.591} C_VEL
LIN {X 0,Y 396.098,Z 459.802,A -85,B 0,C 180,E1 -11392.965,E2 -11392.965} C_VEL
LIN {X 0,Y 396.482,Z 454.159,A -85,B 0,C 180,E1 -11394.609,E2 -11394.609} C_VEL
LIN {X 0,Y 396.995,Z 446.769,A -85,B 0,C 180,E1 -11396.291,E2 -11396.291} C_VEL
LIN {X 0,Y 397.56,Z 439.202,A -85,B 0,C 180,E1 -11397.675,E2 -11397.675} C_VEL
LIN {X 0,Y 398.292,Z 429.743,A -85,B 0,C 180,E1 -11399.077,E2 -11399.077} C_VEL
LIN {X 0,Y 399.139,Z 419.111,A -85,B 0,C 180,E1 -11400.337,E2 -11400.337} C_VEL
LIN {X 0,Y 399.941,Z 407.825,A -85,B 0,C 180,E1 -11401.407,E2 -11401.407} C_VEL
LIN {X 0,Y 400.607,Z 396.772,A -85,B 0,C 180,E1 -11402.228,E2 -11402.228} C_VEL
LIN {X 0,Y 401.269,Z 383.77,A -85,B 0,C 180,E1 -11402.959,E2 -11402.959} C_VEL
LIN {X 0,Y 401.746,Z 370.558,A -85,B 0,C 180,E1 -11403.476,E2 -11403.476} C_VEL
LIN {X 0,Y 402.166,Z 353.586,A -85,B 0,C 180,E1 -11403.854,E2 -11403.854} C_VEL
LIN {X 0,Y 403.179,Z 282.081,A -85,B 0,C 180,E1 -11405.203,E2 -11405.203} C_VEL
LIN {X 0,Y 399.08,Z 259.27,A -85,B 0,C 180,E1 -11405.867,E2 -11405.867} C_VEL
LIN {X 0,Y 399.325,Z 255.278,A -85,B 0,C 180,E1 -11406.746,E2 -11406.746} C_VEL
LIN {X 0,Y 399.458,Z 249.919,A -85,B 0,C 180,E1 -11408.048,E2 -11408.048} C_VEL
LIN {X 0,Y 397.153,Z 237.735,A -85,B 0,C 180,E1 -11411.228,E2 -11411.228} C_VEL
LIN {X 0,Y 397.104,Z 237.518,A -85,B 0,C 180,E1 -11413.553,E2 -11413.553} C_VEL
LIN {X 0,Y 397.107,Z 237.518,A -85,B 0,C 180,E1 -11414.97,E2 -11414.97} C_VEL
LIN {X 0,Y 396.428,Z 237.602,A -85,B 0,C 180,E1 -11415.816,E2 -11415.816} C_VEL
LIN {X 0,Y 393.562,Z 237.958,A -85,B 0,C 180,E1 -11417.193,E2 -11417.193} C_VEL
LIN {X 0,Y 391.161,Z 238.259,A -85,B 0,C 180,E1 -11418.304,E2 -11418.304} C_VEL
LIN {X 0,Y 390.161,Z 238.382,A -85,B 0,C 180,E1 -11419.164,E2 -11419.164} C_VEL
LIN {X 0,Y 390.096,Z 238.388,A -85,B 0,C 180,E1 -11419.455,E2 -11419.455} C_VEL
LIN {X 0,Y 390.234,Z 238.379,A -85,B 0,C 180,E1 -11422.759,E2 -11422.759} C_VEL
LIN {X 0,Y 390.163,Z 238.388,A -85,B 0,C 180,E1 -11424.835,E2 -11424.835} C_VEL
LIN {X 0,Y 390.349,Z 238.357,A -85,B 0,C 180,E1 -11427.938,E2 -11427.938} C_VEL
LIN {X 0,Y 390.478,Z 238.341,A -85,B 0,C 180,E1 -11430.002,E2 -11430.002} C_VEL
LIN {X 0,Y 390.279,Z 238.373,A -85,B 0,C 180,E1 -11433.099,E2 -11433.099} C_VEL
LIN {X 0,Y 390.266,Z 238.367,A -85,B 0,C 180,E1 -11436.205,E2 -11436.205} C_VEL
LIN {X 0,Y 390.141,Z 238.391,A -85,B 0,C 180,E1 -11439.332,E2 -11439.332} C_VEL
LIN {X 0,Y 390.111,Z 238.387,A -85,B 0,C 180,E1 -11442.487,E2 -11442.487} C_VEL
LIN {X 0,Y 390.073,Z 238.397,A -85,B 0,C 180,E1 -11445.681,E2 -11445.681} C_VEL
LIN {X 0,Y 390.039,Z 238.396,A -85,B 0,C 180,E1 -11448.927,E2 -11448.927} C_VEL
LIN {X 0,Y 389.976,Z 238.405,A -85,B 0,C 180,E1 -11452.24,E2 -11452.24} C_VEL
LIN {X 0,Y 390.059,Z 238.399,A -85,B 0,C 180,E1 -11455.749,E2 -11455.749} C_VEL
LIN {X 0,Y 390.007,Z 238.4,A -85,B 0,C 180,E1 -11459.115,E2 -11459.115} C_VEL
LIN {X 0,Y 390.002,Z 238.401,A -85,B 0,C 180,E1 -11462.727,E2 -11462.727} C_VEL
LIN {X 0,Y 390.006,Z 238.402,A -85,B 0,C 180,E1 -11465.832,E2 -11465.832} C_VEL
LIN {X 0,Y 390.026,Z 238.397,A -85,B 0,C 180,E1 -11469.226,E2 -11469.226} C_VEL
LIN {X 0,Y 390.076,Z 238.398,A -85,B 0,C 180,E1 -11472.394,E2 -11472.394} C_VEL
LIN {X 0,Y 390.089,Z 238.391,A -85,B 0,C 180,E1 -11476.11,E2 -11476.11} C_VEL
LIN {X 0,Y 390.042,Z 238.395,A -85,B 0,C 180,E1 -11479.571,E2 -11479.571} C_VEL
LIN {X 0,Y 390.027,Z 238.4,A -85,B 0,C 180,E1 -11482.454,E2 -11482.454} C_VEL
LIN {X 0,Y 390.039,Z 238.396,A -85,B 0,C 180,E1 -11486.053,E2 -11486.053} C_VEL
LIN {X 0,Y 390.021,Z 238.398,A -85,B 0,C 180,E1 -11489.878,E2 -11489.878} C_VEL
LIN {X 0,Y 390.093,Z 238.395,A -85,B 0,C 180,E1 -11493.24,E2 -11493.24} C_VEL
LIN {X 0,Y 390.052,Z 238.396,A -85,B 0,C 180,E1 -11496.772,E2 -11496.772} C_VEL
LIN {X 0,Y 390.091,Z 238.39,A -85,B 0,C 180,E1 -11499.991,E2 -11499.991} C_VEL
LIN {X 0,Y 390.129,Z 238.389,A -85,B 0,C 180,E1 -11503.256,E2 -11503.256} C_VEL
LIN {X 0,Y 390.189,Z 238.377,A -85,B 0,C 180,E1 -11506.569,E2 -11506.569} C_VEL
LIN {X 0,Y 390.163,Z 238.387,A -85,B 0,C 180,E1 -11509.63,E2 -11509.63} C_VEL
LIN {X 0,Y 390.248,Z 238.369,A -85,B 0,C 180,E1 -11512.765,E2 -11512.765} C_VEL
LIN {X 0,Y 390.211,Z 238.374,A -85,B 0,C 180,E1 -11514.84,E2 -11514.84} C_VEL
LIN {X 0,Y 390.417,Z 238.355,A -85,B 0,C 180,E1 -11517.944,E2 -11517.944} C_VEL
LIN {X 0,Y 390.414,Z 238.356,A -85,B 0,C 180,E1 -11522.07,E2 -11522.07} C_VEL
LIN {X 0,Y 390.293,Z 238.371,A -85,B 0,C 180,E1 -11526.209,E2 -11526.209} C_VEL
LIN {X 0,Y 390.2,Z 238.375,A -85,B 0,C 180,E1 -11529.335,E2 -11529.335} C_VEL
LIN {X 0,Y 390.184,Z 238.385,A -85,B 0,C 180,E1 -11532.489,E2 -11532.489} C_VEL
LIN {X 0,Y 390.154,Z 238.381,A -85,B 0,C 180,E1 -11535.682,E2 -11535.682} C_VEL
LIN {X 0,Y 390.12,Z 238.39,A -85,B 0,C 180,E1 -11538.927,E2 -11538.927} C_VEL
LIN {X 0,Y 390.054,Z 238.395,A -85,B 0,C 180,E1 -11542.239,E2 -11542.239} C_VEL
LIN {X 0,Y 390.071,Z 238.392,A -85,B 0,C 180,E1 -11545.726,E2 -11545.726} C_VEL
LIN {X 0,Y 390.045,Z 238.402,A -85,B 0,C 180,E1 -11549.116,E2 -11549.116} C_VEL
LIN {X 0,Y 390.063,Z 238.395,A -85,B 0,C 180,E1 -11552.725,E2 -11552.725} C_VEL
LIN {X 0,Y 390.075,Z 238.393,A -85,B 0,C 180,E1 -11555.827,E2 -11555.827} C_VEL
LIN {X 0,Y 390.06,Z 238.398,A -85,B 0,C 180,E1 -11559.215,E2 -11559.215} C_VEL
LIN {X 0,Y 390.029,Z 238.397,A -85,B 0,C 180,E1 -11562.37,E2 -11562.37} C_VEL
LIN {X 0,Y 390.03,Z 238.401,A -85,B 0,C 180,E1 -11565.351,E2 -11565.351} C_VEL
LIN {X 0,Y 390.026,Z 238.399,A -85,B 0,C 180,E1 -11568.184,E2 -11568.184} C_VEL
LIN {X 0,Y 390.079,Z 238.39,A -85,B 0,C 180,E1 -11570.905,E2 -11570.905} C_VEL
LIN {X 0,Y 390.093,Z 238.389,A -85,B 0,C 180,E1 -11574.792,E2 -11574.792} C_VEL
LIN {X 0,Y 390.044,Z 238.401,A -85,B 0,C 180,E1 -11578.496,E2 -11578.496} C_VEL
LIN {X 0,Y 390.059,Z 238.4,A -85,B 0,C 180,E1 -11582.064,E2 -11582.064} C_VEL
LIN {X 0,Y 390.149,Z 238.594,A -85,B 0,C 180,E1 -11582.581,E2 -11582.581} C_VEL
LIN {X 0,Y 392.36,Z 249.783,A -85,B 0,C 180,E1 -11585.387,E2 -11585.387} C_VEL
LIN {X 0,Y 393.119,Z 254.746,A -85,B 0,C 180,E1 -11586.583,E2 -11586.583} C_VEL
LIN {X 0,Y 392.013,Z 269.033,A -85,B 0,C 180,E1 -11589.776,E2 -11589.776} C_VEL
LIN {X 0,Y 392.335,Z 271.696,A -85,B 0,C 180,E1 -11589.923,E2 -11589.923} C_VEL
LIN {X 0,Y 396.368,Z 296.657,A -85,B 0,C 180,E1 -11590.608,E2 -11590.608} C_VEL
LIN {X 0,Y 395.069,Z 377.738,A -85,B 0,C 180,E1 -11592.195,E2 -11592.195} C_VEL
LIN {X 0,Y 394.539,Z 391.304,A -85,B 0,C 180,E1 -11592.672,E2 -11592.672} C_VEL
LIN {X 0,Y 393.909,Z 403.101,A -85,B 0,C 180,E1 -11593.278,E2 -11593.278} C_VEL
LIN {X 0,Y 393.097,Z 414.319,A -85,B 0,C 180,E1 -11594.043,E2 -11594.043} C_VEL
LIN {X 0,Y 392.293,Z 425.985,A -85,B 0,C 180,E1 -11595.075,E2 -11595.075} C_VEL
LIN {X 0,Y 391.476,Z 436.906,A -85,B 0,C 180,E1 -11596.288,E2 -11596.288} C_VEL
LIN {X 0,Y 390.741,Z 445.941,A -85,B 0,C 180,E1 -11597.534,E2 -11597.534} C_VEL
LIN {X 0,Y 389.949,Z 455.058,A -85,B 0,C 180,E1 -11599.09,E2 -11599.09} C_VEL
LIN {X 0,Y 389.446,Z 462.401,A -85,B 0,C 180,E1 -11600.651,E2 -11600.651} C_VEL
LIN {X 0,Y 389.063,Z 468.26,A -85,B 0,C 180,E1 -11602.212,E2 -11602.212} C_VEL
LIN {X 0,Y 388.817,Z 472.977,A -85,B 0,C 180,E1 -11603.822,E2 -11603.822} C_VEL
LIN {X 0,Y 388.763,Z 475.271,A -85,B 0,C 180,E1 -11604.812,E2 -11604.812} C_VEL
LIN {X 0,Y 388.701,Z 477.245,A -85,B 0,C 180,E1 -11605.851,E2 -11605.851} C_VEL
LIN {X 0,Y 388.609,Z 478.797,A -85,B 0,C 180,E1 -11606.888,E2 -11606.888} C_VEL
LIN {X 0,Y 388.625,Z 479.888,A -85,B 0,C 180,E1 -11607.926,E2 -11607.926} C_VEL
LIN {X 0,Y 388.664,Z 480.57,A -85,B 0,C 180,E1 -11608.962,E2 -11608.962} C_VEL
LIN {X 0,Y 388.681,Z 480.86,A -85,B 0,C 180,E1 -11609.998,E2 -11609.998} C_VEL
LIN {X 0,Y 388.663,Z 480.752,A -85,B 0,C 180,E1 -11611.034,E2 -11611.034} C_VEL
LIN {X 0,Y 388.623,Z 480.202,A -85,B 0,C 180,E1 -11612.071,E2 -11612.071} C_VEL
LIN {X 0,Y 388.706,Z 477.901,A -85,B 0,C 180,E1 -11614.146,E2 -11614.146} C_VEL
LIN {X 0,Y 388.784,Z 474.827,A -85,B 0,C 180,E1 -11615.808,E2 -11615.808} C_VEL
LIN {X 0,Y 389.017,Z 471.149,A -85,B 0,C 180,E1 -11617.263,E2 -11617.263} C_VEL
LIN {X 0,Y 389.373,Z 466.117,A -85,B 0,C 180,E1 -11618.823,E2 -11618.823} C_VEL
LIN {X 0,Y 389.895,Z 459.796,A -85,B 0,C 180,E1 -11620.383,E2 -11620.383} C_VEL
LIN {X 0,Y 390.575,Z 451.887,A -85,B 0,C 180,E1 -11621.941,E2 -11621.941} C_VEL
LIN {X 0,Y 391.651,Z 442.029,A -85,B 0,C 180,E1 -11623.488,E2 -11623.488} C_VEL
LIN {X 0,Y 392.474,Z 432.026,A -85,B 0,C 180,E1 -11624.755,E2 -11624.755} C_VEL
LIN {X 0,Y 393.316,Z 421.686,A -85,B 0,C 180,E1 -11625.811,E2 -11625.811} C_VEL
LIN {X 0,Y 394.252,Z 410.707,A -85,B 0,C 180,E1 -11626.703,E2 -11626.703} C_VEL
LIN {X 0,Y 395.035,Z 399.728,A -85,B 0,C 180,E1 -11627.402,E2 -11627.402} C_VEL
LIN {X 0,Y 395.715,Z 387.005,A -85,B 0,C 180,E1 -11628.005,E2 -11628.005} C_VEL
LIN {X 0,Y 396.252,Z 373.392,A -85,B 0,C 180,E1 -11628.415,E2 -11628.415} C_VEL
LIN {X 0,Y 397.581,Z 296.708,A -85,B 0,C 180,E1 -11629.932,E2 -11629.932} C_VEL
LIN {X 0,Y 394.079,Z 275.978,A -85,B 0,C 180,E1 -11630.583,E2 -11630.583} C_VEL
LIN {X 0,Y 392.555,Z 268.552,A -85,B 0,C 180,E1 -11630.862,E2 -11630.862} C_VEL
LIN {X 0,Y 393.44,Z 255.485,A -85,B 0,C 180,E1 -11633.696,E2 -11633.696} C_VEL
LIN {X 0,Y 391.506,Z 244.616,A -85,B 0,C 180,E1 -11636.336,E2 -11636.336} C_VEL
LIN {X 0,Y 390.136,Z 238.462,A -85,B 0,C 180,E1 -11637.962,E2 -11637.962} C_VEL
LIN {X 0,Y 390.033,Z 238.401,A -85,B 0,C 180,E1 -11641.501,E2 -11641.501} C_VEL
LIN {X 0,Y 390.093,Z 238.393,A -85,B 0,C 180,E1 -11645.203,E2 -11645.203} C_VEL
LIN {X 0,Y 390.065,Z 238.395,A -85,B 0,C 180,E1 -11649.092,E2 -11649.092} C_VEL
LIN {X 0,Y 390.037,Z 238.401,A -85,B 0,C 180,E1 -11652.367,E2 -11652.367} C_VEL
LIN {X 0,Y 390.045,Z 238.396,A -85,B 0,C 180,E1 -11655.349,E2 -11655.349} C_VEL
LIN {X 0,Y 390.019,Z 238.401,A -85,B 0,C 180,E1 -11658.18,E2 -11658.18} C_VEL
LIN {X 0,Y 390.06,Z 238.395,A -85,B 0,C 180,E1 -11660.899,E2 -11660.899} C_VEL
LIN {X 0,Y 390.07,Z 238.397,A -85,B 0,C 180,E1 -11664.786,E2 -11664.786} C_VEL
LIN {X 0,Y 390.023,Z 238.405,A -85,B 0,C 180,E1 -11668.49,E2 -11668.49} C_VEL
LIN {X 0,Y 390.015,Z 238.402,A -85,B 0,C 180,E1 -11671.997,E2 -11671.997} C_VEL
LIN {X 0,Y 390.038,Z 238.398,A -85,B 0,C 180,E1 -11675.511,E2 -11675.511} C_VEL
LIN {X 0,Y 390.045,Z 238.402,A -85,B 0,C 180,E1 -11678.871,E2 -11678.871} C_VEL
LIN {X 0,Y 390.065,Z 238.399,A -85,B 0,C 180,E1 -11682.723,E2 -11682.723} C_VEL
LIN {X 0,Y 390.164,Z 238.385,A -85,B 0,C 180,E1 -11686.57,E2 -11686.57} C_VEL
LIN {X 0,Y 390.15,Z 238.385,A -85,B 0,C 180,E1 -11689.616,E2 -11689.616} C_VEL
LIN {X 0,Y 390.265,Z 238.372,A -85,B 0,C 180,E1 -11692.752,E2 -11692.752} C_VEL
LIN {X 0,Y 390.195,Z 238.377,A -85,B 0,C 180,E1 -11694.827,E2 -11694.827} C_VEL
LIN {X 0,Y 390.392,Z 238.354,A -85,B 0,C 180,E1 -11697.93,E2 -11697.93} C_VEL
LIN {X 0,Y 390.528,Z 238.335,A -85,B 0,C 180,E1 -11699.993,E2 -11699.993} C_VEL
LIN {X 0,Y 390.289,Z 238.367,A -85,B 0,C 180,E1 -11703.09,E2 -11703.09} C_VEL
LIN {X 0,Y 390.264,Z 238.37,A -85,B 0,C 180,E1 -11706.46,E2 -11706.46} C_VEL
LIN {X 0,Y 390.184,Z 238.383,A -85,B 0,C 180,E1 -11709.322,E2 -11709.322} C_VEL
LIN {X 0,Y 390.151,Z 238.385,A -85,B 0,C 180,E1 -11712.476,E2 -11712.476} C_VEL
LIN {X 0,Y 390.11,Z 238.394,A -85,B 0,C 180,E1 -11715.67,E2 -11715.67} C_VEL
LIN {X 0,Y 390.085,Z 238.395,A -85,B 0,C 180,E1 -11718.915,E2 -11718.915} C_VEL
LIN {X 0,Y 390.16,Z 238.577,A -85,B 0,C 180,E1 -11720.527,E2 -11720.527} C_VEL
LIN {X 0,Y 392.744,Z 250.528,A -85,B 0,C 180,E1 -11723.444,E2 -11723.444} C_VEL
LIN {X 0,Y 393.041,Z 254.206,A -85,B 0,C 180,E1 -11724.275,E2 -11724.275} C_VEL
LIN {X 0,Y 392.757,Z 258.507,A -85,B 0,C 180,E1 -11725.176,E2 -11725.176} C_VEL
LIN {X 0,Y 394.73,Z 267.56,A -85,B 0,C 180,E1 -11725.53,E2 -11725.53} C_VEL
LIN {X 0,Y 397.819,Z 283.637,A -85,B 0,C 180,E1 -11726.06,E2 -11726.06} C_VEL
LIN {X 0,Y 396.198,Z 367.409,A -85,B 0,C 180,E1 -11727.733,E2 -11727.733} C_VEL
LIN {X 0,Y 395.628,Z 381.006,A -85,B 0,C 180,E1 -11728.217,E2 -11728.217} C_VEL
LIN {X 0,Y 394.988,Z 393.784,A -85,B 0,C 180,E1 -11728.897,E2 -11728.897} C_VEL
LIN {X 0,Y 394.091,Z 405.552,A -85,B 0,C 180,E1 -11729.735,E2 -11729.735} C_VEL
LIN {X 0,Y 393.143,Z 417.128,A -85,B 0,C 180,E1 -11730.795,E2 -11730.795} C_VEL
LIN {X 0,Y 392.257,Z 426.759,A -85,B 0,C 180,E1 -11731.897,E2 -11731.897} C_VEL
LIN {X 0,Y 391.445,Z 435.943,A -85,B 0,C 180,E1 -11733.192,E2 -11733.192} C_VEL
LIN {X 0,Y 390.546,Z 444.333,A -85,B 0,C 180,E1 -11734.637,E2 -11734.637} C_VEL
LIN {X 0,Y 389.932,Z 451.307,A -85,B 0,C 180,E1 -11736.123,E2 -11736.123} C_VEL
LIN {X 0,Y 389.392,Z 457.74,A -85,B 0,C 180,E1 -11737.842,E2 -11737.842} C_VEL
LIN {X 0,Y 389.047,Z 461.746,A -85,B 0,C 180,E1 -11739.205,E2 -11739.205} C_VEL
LIN {X 0,Y 388.699,Z 466.242,A -85,B 0,C 180,E1 -11741.283,E2 -11741.283} C_VEL
LIN {X 0,Y 388.626,Z 467.592,A -85,B 0,C 180,E1 -11742.148,E2 -11742.148} C_VEL
LIN {X 0,Y 388.511,Z 469.245,A -85,B 0,C 180,E1 -11743.652,E2 -11743.652} C_VEL
LIN {X 0,Y 388.453,Z 470.042,A -85,B 0,C 180,E1 -11745.125,E2 -11745.125} C_VEL
LIN {X 0,Y 388.403,Z 470.023,A -85,B 0,C 180,E1 -11746.563,E2 -11746.563} C_VEL
LIN {X 0,Y 388.459,Z 469.218,A -85,B 0,C 180,E1 -11747.982,E2 -11747.982} C_VEL
LIN {X 0,Y 388.586,Z 466.65,A -85,B 0,C 180,E1 -11750.081,E2 -11750.081} C_VEL
LIN {X 0,Y 388.804,Z 463.798,A -85,B 0,C 180,E1 -11751.552,E2 -11751.552} C_VEL
LIN {X 0,Y 389.138,Z 458.762,A -85,B 0,C 180,E1 -11753.419,E2 -11753.419} C_VEL
LIN {X 0,Y 389.519,Z 452.972,A -85,B 0,C 180,E1 -11755.053,E2 -11755.053} C_VEL
LIN {X 0,Y 390.054,Z 445.759,A -85,B 0,C 180,E1 -11756.667,E2 -11756.667} C_VEL
LIN {X 0,Y 390.634,Z 438.475,A -85,B 0,C 180,E1 -11757.984,E2 -11757.984} C_VEL
LIN {X 0,Y 391.348,Z 429.443,A -85,B 0,C 180,E1 -11759.322,E2 -11759.322} C_VEL
LIN {X 0,Y 392.266,Z 418.471,A -85,B 0,C 180,E1 -11760.632,E2 -11760.632} C_VEL
LIN {X 0,Y 393.08,Z 406.926,A -85,B 0,C 180,E1 -11761.721,E2 -11761.721} C_VEL
LIN {X 0,Y 393.868,Z 394.44,A -85,B 0,C 180,E1 -11762.631,E2 -11762.631} C_VEL
LIN {X 0,Y 394.487,Z 381.924,A -85,B 0,C 180,E1 -11763.312,E2 -11763.312} C_VEL
LIN {X 0,Y 395.04,Z 368.349,A -85,B 0,C 180,E1 -11763.807,E2 -11763.807} C_VEL
LIN {X 0,Y 395.465,Z 343.067,A -85,B 0,C 180,E1 -11764.333,E2 -11764.333} C_VEL
LIN {X 0,Y 396.344,Z 282.323,A -85,B 0,C 180,E1 -11765.512,E2 -11765.512} C_VEL
LIN {X 0,Y 392.196,Z 259.584,A -85,B 0,C 180,E1 -11766.182,E2 -11766.182} C_VEL
LIN {X 0,Y 392.175,Z 258.554,A -85,B 0,C 180,E1 -11766.332,E2 -11766.332} C_VEL
LIN {X 0,Y 392.599,Z 251.983,A -85,B 0,C 180,E1 -11767.921,E2 -11767.921} C_VEL
LIN {X 0,Y 390.381,Z 239.925,A -85,B 0,C 180,E1 -11771.094,E2 -11771.094} C_VEL
LIN {X 0,Y 390.101,Z 238.416,A -85,B 0,C 180,E1 -11771.591,E2 -11771.591} C_VEL
LIN {X 0,Y 390.085,Z 238.392,A -85,B 0,C 180,E1 -11775.392,E2 -11775.392} C_VEL
LIN {X 0,Y 390.089,Z 238.396,A -85,B 0,C 180,E1 -11778.571,E2 -11778.571} C_VEL
LIN {X 0,Y 390.096,Z 238.388,A -85,B 0,C 180,E1 -11779.455,E2 -11779.455} C_VEL
LIN {X 0,Y 389.494,Z 238.469,A -85,B 0,C 180,E1 -11780.318,E2 -11780.318} C_VEL
LIN {X 0,Y 386.738,Z 238.807,A -85,B 0,C 180,E1 -11781.722,E2 -11781.722} C_VEL
LIN {X 0,Y 384.35,Z 239.111,A -85,B 0,C 180,E1 -11782.857,E2 -11782.857} C_VEL
LIN {X 0,Y 383.284,Z 239.238,A -85,B 0,C 180,E1 -11783.733,E2 -11783.733} C_VEL
LIN {X 0,Y 383.177,Z 239.251,A -85,B 0,C 180,E1 -11784.029,E2 -11784.029} C_VEL
LIN {X 0,Y 383.318,Z 239.233,A -85,B 0,C 180,E1 -11787.9,E2 -11787.9} C_VEL
LIN {X 0,Y 383.448,Z 239.216,A -85,B 0,C 180,E1 -11790.002,E2 -11790.002} C_VEL
LIN {X 0,Y 383.213,Z 239.253,A -85,B 0,C 180,E1 -11793.156,E2 -11793.156} C_VEL
LIN {X 0,Y 383.221,Z 239.245,A -85,B 0,C 180,E1 -11796.319,E2 -11796.319} C_VEL
LIN {X 0,Y 383.088,Z 239.267,A -85,B 0,C 180,E1 -11799.505,E2 -11799.505} C_VEL
LIN {X 0,Y 383.074,Z 239.264,A -85,B 0,C 180,E1 -11802.72,E2 -11802.72} C_VEL
LIN {X 0,Y 383.014,Z 239.273,A -85,B 0,C 180,E1 -11805.978,E2 -11805.978} C_VEL
LIN {X 0,Y 382.994,Z 239.276,A -85,B 0,C 180,E1 -11809.289,E2 -11809.289} C_VEL
LIN {X 0,Y 382.945,Z 239.279,A -85,B 0,C 180,E1 -11812.67,E2 -11812.67} C_VEL
LIN {X 0,Y 383.021,Z 239.274,A -85,B 0,C 180,E1 -11816.129,E2 -11816.129} C_VEL
LIN {X 0,Y 382.992,Z 239.275,A -85,B 0,C 180,E1 -11818.498,E2 -11818.498} C_VEL
LIN {X 0,Y 382.954,Z 239.282,A -85,B 0,C 180,E1 -11822.433,E2 -11822.433} C_VEL
LIN {X 0,Y 382.975,Z 239.28,A -85,B 0,C 180,E1 -11825.963,E2 -11825.963} C_VEL
LIN {X 0,Y 382.975,Z 239.276,A -85,B 0,C 180,E1 -11829.595,E2 -11829.595} C_VEL
LIN {X 0,Y 383.023,Z 239.273,A -85,B 0,C 180,E1 -11832.796,E2 -11832.796} C_VEL
LIN {X 0,Y 383.032,Z 239.269,A -85,B 0,C 180,E1 -11835.808,E2 -11835.808} C_VEL
LIN {X 0,Y 383.008,Z 239.277,A -85,B 0,C 180,E1 -11838.794,E2 -11838.794} C_VEL
LIN {X 0,Y 382.977,Z 239.276,A -85,B 0,C 180,E1 -11842.103,E2 -11842.103} C_VEL
LIN {X 0,Y 382.989,Z 239.276,A -85,B 0,C 180,E1 -11845.34,E2 -11845.34} C_VEL
LIN {X 0,Y 382.957,Z 239.284,A -85,B 0,C 180,E1 -11849.09,E2 -11849.09} C_VEL
LIN {X 0,Y 383.036,Z 239.27,A -85,B 0,C 180,E1 -11852.706,E2 -11852.706} C_VEL
LIN {X 0,Y 383.033,Z 239.274,A -85,B 0,C 180,E1 -11855.048,E2 -11855.048} C_VEL
LIN {X 0,Y 382.978,Z 239.275,A -85,B 0,C 180,E1 -11858.477,E2 -11858.477} C_VEL
LIN {X 0,Y 383.042,Z 239.27,A -85,B 0,C 180,E1 -11861.834,E2 -11861.834} C_VEL
LIN {X 0,Y 383.102,Z 239.262,A -85,B 0,C 180,E1 -11865.126,E2 -11865.126} C_VEL
LIN {X 0,Y 383.091,Z 239.262,A -85,B 0,C 180,E1 -11868.366,E2 -11868.366} C_VEL
LIN {X 0,Y 383.215,Z 239.25,A -85,B 0,C 180,E1 -11872.036,E2 -11872.036} C_VEL
LIN {X 0,Y 383.182,Z 239.25,A -85,B 0,C 180,E1 -11874.746,E2 -11874.746} C_VEL
LIN {X 0,Y 383.383,Z 239.231,A -85,B 0,C 180,E1 -11877.906,E2 -11877.906} C_VEL
LIN {X 0,Y 383.38,Z 239.232,A -85,B 0,C 180,E1 -11882.108,E2 -11882.108} C_VEL
LIN {X 0,Y 383.25,Z 239.248,A -85,B 0,C 180,E1 -11886.323,E2 -11886.323} C_VEL
LIN {X 0,Y 383.151,Z 239.254,A -85,B 0,C 180,E1 -11889.508,E2 -11889.508} C_VEL
LIN {X 0,Y 383.142,Z 239.255,A -85,B 0,C 180,E1 -11893.542,E2 -11893.542} C_VEL
LIN {X 0,Y 383.111,Z 239.261,A -85,B 0,C 180,E1 -11897.074,E2 -11897.074} C_VEL
LIN {X 0,Y 383.048,Z 239.272,A -85,B 0,C 180,E1 -11900.651,E2 -11900.651} C_VEL
LIN {X 0,Y 383.028,Z 239.269,A -85,B 0,C 180,E1 -11903.813,E2 -11903.813} C_VEL
LIN {X 0,Y 382.99,Z 239.277,A -85,B 0,C 180,E1 -11907.313,E2 -11907.313} C_VEL
LIN {X 0,Y 383.002,Z 239.277,A -85,B 0,C 180,E1 -11910.922,E2 -11910.922} C_VEL
LIN {X 0,Y 383.039,Z 239.269,A -85,B 0,C 180,E1 -11914.671,E2 -11914.671} C_VEL
LIN {X 0,Y 383.016,Z 239.272,A -85,B 0,C 180,E1 -11917.905,E2 -11917.905} C_VEL
LIN {X 0,Y 382.979,Z 239.281,A -85,B 0,C 180,E1 -11921.354,E2 -11921.354} C_VEL
LIN {X 0,Y 382.987,Z 239.274,A -85,B 0,C 180,E1 -11924.3,E2 -11924.3} C_VEL
LIN {X 0,Y 383,Z 239.275,A -85,B 0,C 180,E1 -11927.237,E2 -11927.237} C_VEL
LIN {X 0,Y 383.008,Z 239.272,A -85,B 0,C 180,E1 -11930.421,E2 -11930.421} C_VEL
LIN {X 0,Y 383.036,Z 239.273,A -85,B 0,C 180,E1 -11934.044,E2 -11934.044} C_VEL
LIN {X 0,Y 383.008,Z 239.274,A -85,B 0,C 180,E1 -11937.58,E2 -11937.58} C_VEL
LIN {X 0,Y 383.002,Z 239.279,A -85,B 0,C 180,E1 -11940.299,E2 -11940.299} C_VEL
LIN {X 0,Y 383.066,Z 239.371,A -85,B 0,C 180,E1 -11942.265,E2 -11942.265} C_VEL
LIN {X 0,Y 385.339,Z 250.707,A -85,B 0,C 180,E1 -11945.196,E2 -11945.196} C_VEL
LIN {X 0,Y 386.125,Z 256.787,A -85,B 0,C 180,E1 -11946.678,E2 -11946.678} C_VEL
LIN {X 0,Y 385.093,Z 269.132,A -85,B 0,C 180,E1 -11949.466,E2 -11949.466} C_VEL
LIN {X 0,Y 385.815,Z 273.969,A -85,B 0,C 180,E1 -11949.652,E2 -11949.652} C_VEL
LIN {X 0,Y 389.55,Z 297.04,A -85,B 0,C 180,E1 -11950.302,E2 -11950.302} C_VEL
LIN {X 0,Y 388.247,Z 377.297,A -85,B 0,C 180,E1 -11951.905,E2 -11951.905} C_VEL
LIN {X 0,Y 387.65,Z 390.954,A -85,B 0,C 180,E1 -11952.388,E2 -11952.388} C_VEL
LIN {X 0,Y 387.015,Z 403.37,A -85,B 0,C 180,E1 -11953.039,E2 -11953.039} C_VEL
LIN {X 0,Y 386.133,Z 415.283,A -85,B 0,C 180,E1 -11953.883,E2 -11953.883} C_VEL
LIN {X 0,Y 385.296,Z 426.757,A -85,B 0,C 180,E1 -11954.933,E2 -11954.933} C_VEL
LIN {X 0,Y 384.543,Z 436.68,A -85,B 0,C 180,E1 -11956.064,E2 -11956.064} C_VEL
LIN {X 0,Y 383.774,Z 445.573,A -85,B 0,C 180,E1 -11957.304,E2 -11957.304} C_VEL
LIN {X 0,Y 382.941,Z 454.74,A -85,B 0,C 180,E1 -11958.888,E2 -11958.888} C_VEL
LIN {X 0,Y 382.415,Z 462.125,A -85,B 0,C 180,E1 -11960.478,E2 -11960.478} C_VEL
LIN {X 0,Y 382.01,Z 468.027,A -85,B 0,C 180,E1 -11962.067,E2 -11962.067} C_VEL
LIN {X 0,Y 381.714,Z 473.172,A -85,B 0,C 180,E1 -11963.87,E2 -11963.87} C_VEL
LIN {X 0,Y 381.628,Z 477.081,A -85,B 0,C 180,E1 -11965.774,E2 -11965.774} C_VEL
LIN {X 0,Y 381.523,Z 478.647,A -85,B 0,C 180,E1 -11966.83,E2 -11966.83} C_VEL
LIN {X 0,Y 381.523,Z 479.76,A -85,B 0,C 180,E1 -11967.887,E2 -11967.887} C_VEL
LIN {X 0,Y 381.562,Z 480.454,A -85,B 0,C 180,E1 -11968.943,E2 -11968.943} C_VEL
LIN {X 0,Y 381.582,Z 480.755,A -85,B 0,C 180,E1 -11969.998,E2 -11969.998} C_VEL
LIN {X 0,Y 381.562,Z 480.661,A -85,B 0,C 180,E1 -11971.054,E2 -11971.054} C_VEL
LIN {X 0,Y 381.521,Z 480.129,A -85,B 0,C 180,E1 -11972.11,E2 -11972.11} C_VEL
LIN {X 0,Y 381.636,Z 477.846,A -85,B 0,C 180,E1 -11974.222,E2 -11974.222} C_VEL
LIN {X 0,Y 381.703,Z 476.088,A -85,B 0,C 180,E1 -11975.28,E2 -11975.28} C_VEL
LIN {X 0,Y 381.859,Z 472.568,A -85,B 0,C 180,E1 -11976.869,E2 -11976.869} C_VEL
LIN {X 0,Y 382.175,Z 467.948,A -85,B 0,C 180,E1 -11978.458,E2 -11978.458} C_VEL
LIN {X 0,Y 382.765,Z 460.95,A -85,B 0,C 180,E1 -11980.311,E2 -11980.311} C_VEL
LIN {X 0,Y 383.496,Z 453.396,A -85,B 0,C 180,E1 -11981.896,E2 -11981.896} C_VEL
LIN {X 0,Y 384.339,Z 445.694,A -85,B 0,C 180,E1 -11983.211,E2 -11983.211} C_VEL
LIN {X 0,Y 385.281,Z 435.651,A -85,B 0,C 180,E1 -11984.611,E2 -11984.611} C_VEL
LIN {X 0,Y 386.254,Z 424.679,A -85,B 0,C 180,E1 -11985.837,E2 -11985.837} C_VEL
LIN {X 0,Y 387.315,Z 412.851,A -85,B 0,C 180,E1 -11986.875,E2 -11986.875} C_VEL
LIN {X 0,Y 388.284,Z 400.25,A -85,B 0,C 180,E1 -11987.714,E2 -11987.714} C_VEL
LIN {X 0,Y 389.004,Z 387.781,A -85,B 0,C 180,E1 -11988.327,E2 -11988.327} C_VEL
LIN {X 0,Y 389.56,Z 374.915,A -85,B 0,C 180,E1 -11988.743,E2 -11988.743} C_VEL
LIN {X 0,Y 391.003,Z 297.379,A -85,B 0,C 180,E1 -11990.311,E2 -11990.311} C_VEL
LIN {X 0,Y 387.274,Z 275.764,A -85,B 0,C 180,E1 -11991.017,E2 -11991.017} C_VEL
LIN {X 0,Y 385.72,Z 268.278,A -85,B 0,C 180,E1 -11991.325,E2 -11991.325} C_VEL
LIN {X 0,Y 386.581,Z 258.104,A -85,B 0,C 180,E1 -11993.573,E2 -11993.573} C_VEL
LIN {X 0,Y 385.542,Z 250.752,A -85,B 0,C 180,E1 -11995.362,E2 -11995.362} C_VEL
LIN {X 0,Y 383.438,Z 240.998,A -85,B 0,C 180,E1 -11997.856,E2 -11997.856} C_VEL
LIN {X 0,Y 383.049,Z 239.3,A -85,B 0,C 180,E1 -11998.408,E2 -11998.408} C_VEL
LIN {X 0,Y 383.019,Z 239.276,A -85,B 0,C 180,E1 -12002.146,E2 -12002.146} C_VEL
LIN {X 0,Y 383.028,Z 239.273,A -85,B 0,C 180,E1 -12004.664,E2 -12004.664} C_VEL
LIN {X 0,Y 383.002,Z 239.277,A -85,B 0,C 180,E1 -12007.898,E2 -12007.898} C_VEL
LIN {X 0,Y 382.968,Z 239.278,A -85,B 0,C 180,E1 -12011.346,E2 -12011.346} C_VEL
LIN {X 0,Y 382.995,Z 239.28,A -85,B 0,C 180,E1 -12014.297,E2 -12014.297} C_VEL
LIN {X 0,Y 382.987,Z 239.276,A -85,B 0,C 180,E1 -12017.231,E2 -12017.231} C_VEL
LIN {X 0,Y 382.989,Z 239.276,A -85,B 0,C 180,E1 -12020.414,E2 -12020.414} C_VEL
LIN {X 0,Y 383.015,Z 239.271,A -85,B 0,C 180,E1 -12024.038,E2 -12024.038} C_VEL
LIN {X 0,Y 382.986,Z 239.274,A -85,B 0,C 180,E1 -12027.573,E2 -12027.573} C_VEL
LIN {X 0,Y 382.975,Z 239.276,A -85,B 0,C 180,E1 -12030.293,E2 -12030.293} C_VEL
LIN {X 0,Y 383.002,Z 239.269,A -85,B 0,C 180,E1 -12034.039,E2 -12034.039} C_VEL
LIN {X 0,Y 382.981,Z 239.273,A -85,B 0,C 180,E1 -12037.328,E2 -12037.328} C_VEL
LIN {X 0,Y 383.007,Z 239.272,A -85,B 0,C 180,E1 -12040.708,E2 -12040.708} C_VEL
LIN {X 0,Y 383.003,Z 239.271,A -85,B 0,C 180,E1 -12044.017,E2 -12044.017} C_VEL
LIN {X 0,Y 383.121,Z 239.256,A -85,B 0,C 180,E1 -12047.277,E2 -12047.277} C_VEL
LIN {X 0,Y 383.128,Z 239.26,A -85,B 0,C 180,E1 -12050.491,E2 -12050.491} C_VEL
LIN {X 0,Y 383.246,Z 239.242,A -85,B 0,C 180,E1 -12053.677,E2 -12053.677} C_VEL
LIN {X 0,Y 383.358,Z 239.231,A -85,B 0,C 180,E1 -12057.892,E2 -12057.892} C_VEL
LIN {X 0,Y 383.497,Z 239.21,A -85,B 0,C 180,E1 -12059.993,E2 -12059.993} C_VEL
LIN {X 0,Y 383.226,Z 239.248,A -85,B 0,C 180,E1 -12063.147,E2 -12063.147} C_VEL
LIN {X 0,Y 383.228,Z 239.247,A -85,B 0,C 180,E1 -12066.45,E2 -12066.45} C_VEL
LIN {X 0,Y 383.131,Z 239.263,A -85,B 0,C 180,E1 -12069.495,E2 -12069.495} C_VEL
LIN {X 0,Y 383.114,Z 239.262,A -85,B 0,C 180,E1 -12072.709,E2 -12072.709} C_VEL
LIN {X 0,Y 383.051,Z 239.272,A -85,B 0,C 180,E1 -12075.966,E2 -12075.966} C_VEL
LIN {X 0,Y 383.046,Z 239.27,A -85,B 0,C 180,E1 -12079.276,E2 -12079.276} C_VEL
LIN {X 0,Y 383.096,Z 239.426,A -85,B 0,C 180,E1 -12080.11,E2 -12080.11} C_VEL
LIN {X 0,Y 385.407,Z 250.045,A -85,B 0,C 180,E1 -12082.79,E2 -12082.79} C_VEL
LIN {X 0,Y 386.119,Z 253.389,A -85,B 0,C 180,E1 -12083.596,E2 -12083.596} C_VEL
LIN {X 0,Y 386.004,Z 258.731,A -85,B 0,C 180,E1 -12084.747,E2 -12084.747} C_VEL
LIN {X 0,Y 390.172,Z 278.678,A -85,B 0,C 180,E1 -12085.486,E2 -12085.486} C_VEL
LIN {X 0,Y 391.205,Z 284.275,A -85,B 0,C 180,E1 -12085.673,E2 -12085.673} C_VEL
LIN {X 0,Y 389.554,Z 367.789,A -85,B 0,C 180,E1 -12087.379,E2 -12087.379} C_VEL
LIN {X 0,Y 388.949,Z 381.259,A -85,B 0,C 180,E1 -12087.869,E2 -12087.869} C_VEL
LIN {X 0,Y 388.35,Z 393.043,A -85,B 0,C 180,E1 -12088.5,E2 -12088.5} C_VEL
LIN {X 0,Y 387.47,Z 404.526,A -85,B 0,C 180,E1 -12089.313,E2 -12089.313} C_VEL
LIN {X 0,Y 386.52,Z 415.418,A -85,B 0,C 180,E1 -12090.299,E2 -12090.299} C_VEL
LIN {X 0,Y 385.501,Z 425.911,A -85,B 0,C 180,E1 -12091.483,E2 -12091.483} C_VEL
LIN {X 0,Y 384.593,Z 435.318,A -85,B 0,C 180,E1 -12092.801,E2 -12092.801} C_VEL
LIN {X 0,Y 383.726,Z 443.251,A -85,B 0,C 180,E1 -12094.163,E2 -12094.163} C_VEL
LIN {X 0,Y 383.066,Z 450.175,A -85,B 0,C 180,E1 -12095.616,E2 -12095.616} C_VEL
LIN {X 0,Y 382.454,Z 456.694,A -85,B 0,C 180,E1 -12097.319,E2 -12097.319} C_VEL
LIN {X 0,Y 382.089,Z 460.904,A -85,B 0,C 180,E1 -12098.698,E2 -12098.698} C_VEL
LIN {X 0,Y 381.801,Z 464.319,A -85,B 0,C 180,E1 -12100.098,E2 -12100.098} C_VEL
LIN {X 0,Y 381.575,Z 466.953,A -85,B 0,C 180,E1 -12101.521,E2 -12101.521} C_VEL
LIN {X 0,Y 381.471,Z 468.79,A -85,B 0,C 180,E1 -12102.961,E2 -12102.961} C_VEL
LIN {X 0,Y 381.373,Z 469.894,A -85,B 0,C 180,E1 -12104.435,E2 -12104.435} C_VEL
LIN {X 0,Y 381.335,Z 470.22,A -85,B 0,C 180,E1 -12105.939,E2 -12105.939} C_VEL
LIN {X 0,Y 381.305,Z 469.698,A -85,B 0,C 180,E1 -12107.484,E2 -12107.484} C_VEL
LIN {X 0,Y 381.433,Z 468.259,A -85,B 0,C 180,E1 -12109.048,E2 -12109.048} C_VEL
LIN {X 0,Y 381.581,Z 465.817,A -85,B 0,C 180,E1 -12110.659,E2 -12110.659} C_VEL
LIN {X 0,Y 381.843,Z 461.476,A -85,B 0,C 180,E1 -12112.603,E2 -12112.603} C_VEL
LIN {X 0,Y 382.255,Z 456.223,A -85,B 0,C 180,E1 -12114.323,E2 -12114.323} C_VEL
LIN {X 0,Y 382.653,Z 450.852,A -85,B 0,C 180,E1 -12115.722,E2 -12115.722} C_VEL
LIN {X 0,Y 383.218,Z 443.279,A -85,B 0,C 180,E1 -12117.321,E2 -12117.321} C_VEL
LIN {X 0,Y 384.023,Z 434.092,A -85,B 0,C 180,E1 -12118.871,E2 -12118.871} C_VEL
LIN {X 0,Y 384.88,Z 423.36,A -85,B 0,C 180,E1 -12120.312,E2 -12120.312} C_VEL
LIN {X 0,Y 385.837,Z 412.267,A -85,B 0,C 180,E1 -12121.493,E2 -12121.493} C_VEL
LIN {X 0,Y 386.609,Z 400.413,A -85,B 0,C 180,E1 -12122.485,E2 -12122.485} C_VEL
LIN {X 0,Y 387.338,Z 388.588,A -85,B 0,C 180,E1 -12123.245,E2 -12123.245} C_VEL
LIN {X 0,Y 387.912,Z 375.605,A -85,B 0,C 180,E1 -12123.85,E2 -12123.85} C_VEL
LIN {X 0,Y 388.328,Z 362.455,A -85,B 0,C 180,E1 -12124.24,E2 -12124.24} C_VEL
LIN {X 0,Y 389.53,Z 282.999,A -85,B 0,C 180,E1 -12125.813,E2 -12125.813} C_VEL
LIN {X 0,Y 385.304,Z 259.689,A -85,B 0,C 180,E1 -12126.522,E2 -12126.522} C_VEL
LIN {X 0,Y 385.292,Z 258.839,A -85,B 0,C 180,E1 -12126.628,E2 -12126.628} C_VEL
LIN {X 0,Y 385.574,Z 252.783,A -85,B 0,C 180,E1 -12128.117,E2 -12128.117} C_VEL
LIN {X 0,Y 383.182,Z 239.957,A -85,B 0,C 180,E1 -12131.558,E2 -12131.558} C_VEL
LIN {X 0,Y 383.054,Z 239.296,A -85,B 0,C 180,E1 -12131.828,E2 -12131.828} C_VEL
LIN {X 0,Y 383.05,Z 239.27,A -85,B 0,C 180,E1 -12135.118,E2 -12135.118} C_VEL
LIN {X 0,Y 383.037,Z 239.272,A -85,B 0,C 180,E1 -12138.358,E2 -12138.358} C_VEL
LIN {X 0,Y 383.191,Z 239.249,A -85,B 0,C 180,E1 -12141.975,E2 -12141.975} C_VEL
LIN {X 0,Y 383.177,Z 239.251,A -85,B 0,C 180,E1 -12144.029,E2 -12144.029} C_VEL
LIN {X 0,Y 382.471,Z 239.345,A -85,B 0,C 180,E1 -12144.906,E2 -12144.906} C_VEL
LIN {X 0,Y 379.665,Z 239.689,A -85,B 0,C 180,E1 -12146.334,E2 -12146.334} C_VEL
LIN {X 0,Y 377.32,Z 239.981,A -85,B 0,C 180,E1 -12147.488,E2 -12147.488} C_VEL
LIN {X 0,Y 376.311,Z 240.107,A -85,B 0,C 180,E1 -12148.379,E2 -12148.379} C_VEL
LIN {X 0,Y 376.226,Z 240.12,A -85,B 0,C 180,E1 -12148.681,E2 -12148.681} C_VEL
LIN {X 0,Y 376.418,Z 240.092,A -85,B 0,C 180,E1 -12150.002,E2 -12150.002} C_VEL
LIN {X 0,Y 376.15,Z 240.132,A -85,B 0,C 180,E1 -12153.215,E2 -12153.215} C_VEL
LIN {X 0,Y 376.178,Z 240.123,A -85,B 0,C 180,E1 -12156.438,E2 -12156.438} C_VEL
LIN {X 0,Y 376.055,Z 240.141,A -85,B 0,C 180,E1 -12159.685,E2 -12159.685} C_VEL
LIN {X 0,Y 376.023,Z 240.146,A -85,B 0,C 180,E1 -12163.662,E2 -12163.662} C_VEL
LIN {X 0,Y 375.978,Z 240.155,A -85,B 0,C 180,E1 -12167.611,E2 -12167.611} C_VEL
LIN {X 0,Y 375.916,Z 240.155,A -85,B 0,C 180,E1 -12170.837,E2 -12170.837} C_VEL
LIN {X 0,Y 375.933,Z 240.155,A -85,B 0,C 180,E1 -12174.287,E2 -12174.287} C_VEL
LIN {X 0,Y 375.961,Z 240.15,A -85,B 0,C 180,E1 -12176.658,E2 -12176.658} C_VEL
LIN {X 0,Y 375.92,Z 240.154,A -85,B 0,C 180,E1 -12179.085,E2 -12179.085} C_VEL
LIN {X 0,Y 375.903,Z 240.157,A -85,B 0,C 180,E1 -12182.835,E2 -12182.835} C_VEL
LIN {X 0,Y 375.907,Z 240.156,A -85,B 0,C 180,E1 -12185.423,E2 -12185.423} C_VEL
LIN {X 0,Y 375.929,Z 240.16,A -85,B 0,C 180,E1 -12188.278,E2 -12188.278} C_VEL
LIN {X 0,Y 375.945,Z 240.151,A -85,B 0,C 180,E1 -12191.618,E2 -12191.618} C_VEL
LIN {X 0,Y 375.975,Z 240.148,A -85,B 0,C 180,E1 -12195.263,E2 -12195.263} C_VEL
LIN {X 0,Y 375.965,Z 240.151,A -85,B 0,C 180,E1 -12199.149,E2 -12199.149} C_VEL
LIN {X 0,Y 375.94,Z 240.152,A -85,B 0,C 180,E1 -12201.921,E2 -12201.921} C_VEL
LIN {X 0,Y 375.951,Z 240.153,A -85,B 0,C 180,E1 -12205.341,E2 -12205.341} C_VEL
LIN {X 0,Y 375.931,Z 240.154,A -85,B 0,C 180,E1 -12208.446,E2 -12208.446} C_VEL
LIN {X 0,Y 375.961,Z 240.149,A -85,B 0,C 180,E1 -12212.149,E2 -12212.149} C_VEL
LIN {X 0,Y 375.987,Z 240.147,A -85,B 0,C 180,E1 -12214.547,E2 -12214.547} C_VEL
LIN {X 0,Y 375.942,Z 240.152,A -85,B 0,C 180,E1 -12218.054,E2 -12218.054} C_VEL
LIN {X 0,Y 375.991,Z 240.152,A -85,B 0,C 180,E1 -12221.481,E2 -12221.481} C_VEL
LIN {X 0,Y 376.05,Z 240.139,A -85,B 0,C 180,E1 -12224.841,E2 -12224.841} C_VEL
LIN {X 0,Y 376.044,Z 240.141,A -85,B 0,C 180,E1 -12228.144,E2 -12228.144} C_VEL
LIN {X 0,Y 376.187,Z 240.126,A -85,B 0,C 180,E1 -12231.962,E2 -12231.962} C_VEL
LIN {X 0,Y 376.153,Z 240.126,A -85,B 0,C 180,E1 -12234.647,E2 -12234.647} C_VEL
LIN {X 0,Y 376.348,Z 240.107,A -85,B 0,C 180,E1 -12237.867,E2 -12237.867} C_VEL
LIN {X 0,Y 376.345,Z 240.109,A -85,B 0,C 180,E1 -12242.147,E2 -12242.147} C_VEL
LIN {X 0,Y 376.209,Z 240.124,A -85,B 0,C 180,E1 -12246.442,E2 -12246.442} C_VEL
LIN {X 0,Y 376.122,Z 240.13,A -85,B 0,C 180,E1 -12249.688,E2 -12249.688} C_VEL
LIN {X 0,Y 376.106,Z 240.131,A -85,B 0,C 180,E1 -12253.663,E2 -12253.663} C_VEL
LIN {X 0,Y 376.05,Z 240.139,A -85,B 0,C 180,E1 -12257.405,E2 -12257.405} C_VEL
LIN {X 0,Y 375.998,Z 240.151,A -85,B 0,C 180,E1 -12260.837,E2 -12260.837} C_VEL
LIN {X 0,Y 375.988,Z 240.147,A -85,B 0,C 180,E1 -12264.288,E2 -12264.288} C_VEL
LIN {X 0,Y 375.938,Z 240.152,A -85,B 0,C 180,E1 -12267.869,E2 -12267.869} C_VEL
LIN {X 0,Y 375.977,Z 240.15,A -85,B 0,C 180,E1 -12271.566,E2 -12271.566} C_VEL
LIN {X 0,Y 375.978,Z 240.153,A -85,B 0,C 180,E1 -12275.419,E2 -12275.419} C_VEL
LIN {X 0,Y 375.958,Z 240.15,A -85,B 0,C 180,E1 -12278.265,E2 -12278.265} C_VEL
LIN {X 0,Y 375.932,Z 240.159,A -85,B 0,C 180,E1 -12281.599,E2 -12281.599} C_VEL
LIN {X 0,Y 375.918,Z 240.158,A -85,B 0,C 180,E1 -12285.276,E2 -12285.276} C_VEL
LIN {X 0,Y 375.933,Z 240.153,A -85,B 0,C 180,E1 -12288.406,E2 -12288.406} C_VEL
LIN {X 0,Y 375.975,Z 240.154,A -85,B 0,C 180,E1 -12291.911,E2 -12291.911} C_VEL
LIN {X 0,Y 375.999,Z 240.146,A -85,B 0,C 180,E1 -12295.335,E2 -12295.335} C_VEL
LIN {X 0,Y 375.979,Z 240.154,A -85,B 0,C 180,E1 -12298.438,E2 -12298.438} C_VEL
LIN {X 0,Y 376.009,Z 240.301,A -85,B 0,C 180,E1 -12302.033,E2 -12302.033} C_VEL
LIN {X 0,Y 378.427,Z 252.239,A -85,B 0,C 180,E1 -12305.153,E2 -12305.153} C_VEL
LIN {X 0,Y 379.161,Z 257.702,A -85,B 0,C 180,E1 -12306.513,E2 -12306.513} C_VEL
LIN {X 0,Y 378.186,Z 268.957,A -85,B 0,C 180,E1 -12309.109,E2 -12309.109} C_VEL
LIN {X 0,Y 378.911,Z 273.822,A -85,B 0,C 180,E1 -12309.301,E2 -12309.301} C_VEL
LIN {X 0,Y 382.805,Z 298.404,A -85,B 0,C 180,E1 -12310.013,E2 -12310.013} C_VEL
LIN {X 0,Y 381.403,Z 377.965,A -85,B 0,C 180,E1 -12311.639,E2 -12311.639} C_VEL
LIN {X 0,Y 380.795,Z 391.367,A -85,B 0,C 180,E1 -12312.13,E2 -12312.13} C_VEL
LIN {X 0,Y 380.127,Z 403.624,A -85,B 0,C 180,E1 -12312.792,E2 -12312.792} C_VEL
LIN {X 0,Y 379.166,Z 416.246,A -85,B 0,C 180,E1 -12313.717,E2 -12313.717} C_VEL
LIN {X 0,Y 378.294,Z 427.529,A -85,B 0,C 180,E1 -12314.785,E2 -12314.785} C_VEL
LIN {X 0,Y 377.486,Z 437.686,A -85,B 0,C 180,E1 -12315.992,E2 -12315.992} C_VEL
LIN {X 0,Y 376.651,Z 446.855,A -85,B 0,C 180,E1 -12317.334,E2 -12317.334} C_VEL
LIN {X 0,Y 375.826,Z 455.795,A -85,B 0,C 180,E1 -12318.948,E2 -12318.948} C_VEL
LIN {X 0,Y 375.283,Z 462.942,A -85,B 0,C 180,E1 -12320.567,E2 -12320.567} C_VEL
LIN {X 0,Y 374.827,Z 469.453,A -85,B 0,C 180,E1 -12322.456,E2 -12322.456} C_VEL
LIN {X 0,Y 374.609,Z 473.374,A -85,B 0,C 180,E1 -12323.924,E2 -12323.924} C_VEL
LIN {X 0,Y 374.535,Z 476.916,A -85,B 0,C 180,E1 -12325.694,E2 -12325.694} C_VEL
LIN {X 0,Y 374.441,Z 478.496,A -85,B 0,C 180,E1 -12326.77,E2 -12326.77} C_VEL
LIN {X 0,Y 374.423,Z 479.632,A -85,B 0,C 180,E1 -12327.847,E2 -12327.847} C_VEL
LIN {X 0,Y 374.461,Z 480.338,A -85,B 0,C 180,E1 -12328.923,E2 -12328.923} C_VEL
LIN {X 0,Y 374.483,Z 480.65,A -85,B 0,C 180,E1 -12329.998,E2 -12329.998} C_VEL
LIN {X 0,Y 374.46,Z 480.568,A -85,B 0,C 180,E1 -12331.074,E2 -12331.074} C_VEL
LIN {X 0,Y 374.421,Z 480.056,A -85,B 0,C 180,E1 -12332.15,E2 -12332.15} C_VEL
LIN {X 0,Y 374.544,Z 477.791,A -85,B 0,C 180,E1 -12334.303,E2 -12334.303} C_VEL
LIN {X 0,Y 374.654,Z 474.531,A -85,B 0,C 180,E1 -12336.142,E2 -12336.142} C_VEL
LIN {X 0,Y 375.014,Z 469.606,A -85,B 0,C 180,E1 -12338.078,E2 -12338.078} C_VEL
LIN {X 0,Y 375.569,Z 463.191,A -85,B 0,C 180,E1 -12339.966,E2 -12339.966} C_VEL
LIN {X 0,Y 376.217,Z 456.209,A -85,B 0,C 180,E1 -12341.583,E2 -12341.583} C_VEL
LIN {X 0,Y 377.247,Z 447.467,A -85,B 0,C 180,E1 -12343.19,E2 -12343.19} C_VEL
LIN {X 0,Y 378.265,Z 437.811,A -85,B 0,C 180,E1 -12344.624,E2 -12344.624} C_VEL
LIN {X 0,Y 379.161,Z 427.769,A -85,B 0,C 180,E1 -12345.837,E2 -12345.837} C_VEL
LIN {X 0,Y 380.291,Z 416.398,A -85,B 0,C 180,E1 -12346.92,E2 -12346.92} C_VEL
LIN {X 0,Y 381.271,Z 403.996,A -85,B 0,C 180,E1 -12347.843,E2 -12347.843} C_VEL
LIN {X 0,Y 382.183,Z 391.487,A -85,B 0,C 180,E1 -12348.527,E2 -12348.527} C_VEL
LIN {X 0,Y 382.776,Z 378.517,A -85,B 0,C 180,E1 -12349.018,E2 -12349.018} C_VEL
LIN {X 0,Y 383.36,Z 357.242,A -85,B 0,C 180,E1 -12349.487,E2 -12349.487} C_VEL
LIN {X 0,Y 384.427,Z 297.787,A -85,B 0,C 180,E1 -12350.718,E2 -12350.718} C_VEL
LIN {X 0,Y 380.831,Z 277.145,A -85,B 0,C 180,E1 -12351.418,E2 -12351.418} C_VEL
LIN {X 0,Y 378.936,Z 268.344,A -85,B 0,C 180,E1 -12351.771,E2 -12351.771} C_VEL
LIN {X 0,Y 379.7,Z 259.521,A -85,B 0,C 180,E1 -12353.737,E2 -12353.737} C_VEL
LIN {X 0,Y 378.628,Z 252.165,A -85,B 0,C 180,E1 -12355.564,E2 -12355.564} C_VEL
LIN {X 0,Y 376.474,Z 242.22,A -85,B 0,C 180,E1 -12358.171,E2 -12358.171} C_VEL
LIN {X 0,Y 375.98,Z 240.186,A -85,B 0,C 180,E1 -12358.811,E2 -12358.811} C_VEL
LIN {X 0,Y 375.968,Z 240.154,A -85,B 0,C 180,E1 -12361.558,E2 -12361.558} C_VEL
LIN {X 0,Y 375.966,Z 240.155,A -85,B 0,C 180,E1 -12365.412,E2 -12365.412} C_VEL
LIN {X 0,Y 375.944,Z 240.158,A -85,B 0,C 180,E1 -12368.258,E2 -12368.258} C_VEL
LIN {X 0,Y 375.921,Z 240.157,A -85,B 0,C 180,E1 -12371.592,E2 -12371.592} C_VEL
LIN {X 0,Y 375.926,Z 240.156,A -85,B 0,C 180,E1 -12374.725,E2 -12374.725} C_VEL
LIN {X 0,Y 375.913,Z 240.158,A -85,B 0,C 180,E1 -12377.691,E2 -12377.691} C_VEL
LIN {X 0,Y 375.938,Z 240.154,A -85,B 0,C 180,E1 -12380.529,E2 -12380.529} C_VEL
LIN {X 0,Y 375.96,Z 240.149,A -85,B 0,C 180,E1 -12383.492,E2 -12383.492} C_VEL
LIN {X 0,Y 375.96,Z 240.153,A -85,B 0,C 180,E1 -12385.883,E2 -12385.883} C_VEL
LIN {X 0,Y 375.962,Z 240.149,A -85,B 0,C 180,E1 -12389.681,E2 -12389.681} C_VEL
LIN {X 0,Y 375.917,Z 240.159,A -85,B 0,C 180,E1 -12392.129,E2 -12392.129} C_VEL
LIN {X 0,Y 375.965,Z 240.151,A -85,B 0,C 180,E1 -12395.711,E2 -12395.711} C_VEL
LIN {X 0,Y 375.953,Z 240.154,A -85,B 0,C 180,E1 -12399.189,E2 -12399.189} C_VEL
LIN {X 0,Y 375.974,Z 240.153,A -85,B 0,C 180,E1 -12402.591,E2 -12402.591} C_VEL
LIN {X 0,Y 376.096,Z 240.136,A -85,B 0,C 180,E1 -12406.328,E2 -12406.328} C_VEL
LIN {X 0,Y 376.099,Z 240.135,A -85,B 0,C 180,E1 -12410.312,E2 -12410.312} C_VEL
LIN {X 0,Y 376.205,Z 240.119,A -85,B 0,C 180,E1 -12413.558,E2 -12413.558} C_VEL
LIN {X 0,Y 376.323,Z 240.107,A -85,B 0,C 180,E1 -12417.853,E2 -12417.853} C_VEL
LIN {X 0,Y 376.467,Z 240.086,A -85,B 0,C 180,E1 -12419.993,E2 -12419.993} C_VEL
LIN {X 0,Y 376.164,Z 240.128,A -85,B 0,C 180,E1 -12423.206,E2 -12423.206} C_VEL
LIN {X 0,Y 376.197,Z 240.123,A -85,B 0,C 180,E1 -12426.437,E2 -12426.437} C_VEL
LIN {X 0,Y 376.099,Z 240.14,A -85,B 0,C 180,E1 -12429.674,E2 -12429.674} C_VEL
LIN {X 0,Y 376.061,Z 240.142,A -85,B 0,C 180,E1 -12433.651,E2 -12433.651} C_VEL
LIN {X 0,Y 376.03,Z 240.143,A -85,B 0,C 180,E1 -12437.609,E2 -12437.609} C_VEL
LIN {X 0,Y 376.032,Z 240.377,A -85,B 0,C 180,E1 -12439.721,E2 -12439.721} C_VEL
LIN {X 0,Y 378.331,Z 250.679,A -85,B 0,C 180,E1 -12442.375,E2 -12442.375} C_VEL
LIN {X 0,Y 379.331,Z 256.338,A -85,B 0,C 180,E1 -12443.755,E2 -12443.755} C_VEL
LIN {X 0,Y 379.266,Z 259.055,A -85,B 0,C 180,E1 -12444.304,E2 -12444.304} C_VEL
LIN {X 0,Y 383.834,Z 280.557,A -85,B 0,C 180,E1 -12445.114,E2 -12445.114} C_VEL
LIN {X 0,Y 384.705,Z 286.265,A -85,B 0,C 180,E1 -12445.298,E2 -12445.298} C_VEL
LIN {X 0,Y 382.931,Z 368.006,A -85,B 0,C 180,E1 -12447.006,E2 -12447.006} C_VEL
LIN {X 0,Y 382.286,Z 381.511,A -85,B 0,C 180,E1 -12447.509,E2 -12447.509} C_VEL
LIN {X 0,Y 381.558,Z 394.447,A -85,B 0,C 180,E1 -12448.228,E2 -12448.228} C_VEL
LIN {X 0,Y 380.558,Z 406.645,A -85,B 0,C 180,E1 -12449.139,E2 -12449.139} C_VEL
LIN {X 0,Y 379.609,Z 417.091,A -85,B 0,C 180,E1 -12450.134,E2 -12450.134} C_VEL
LIN {X 0,Y 378.535,Z 427.365,A -85,B 0,C 180,E1 -12451.35,E2 -12451.35} C_VEL
LIN {X 0,Y 377.502,Z 437.483,A -85,B 0,C 180,E1 -12452.856,E2 -12452.856} C_VEL
LIN {X 0,Y 376.54,Z 445.813,A -85,B 0,C 180,E1 -12454.389,E2 -12454.389} C_VEL
LIN {X 0,Y 375.877,Z 452.491,A -85,B 0,C 180,E1 -12455.916,E2 -12455.916} C_VEL
LIN {X 0,Y 375.252,Z 458.891,A -85,B 0,C 180,E1 -12457.777,E2 -12457.777} C_VEL
LIN {X 0,Y 374.777,Z 464.016,A -85,B 0,C 180,E1 -12459.753,E2 -12459.753} C_VEL
LIN {X 0,Y 374.497,Z 466.984,A -85,B 0,C 180,E1 -12461.356,E2 -12461.356} C_VEL
LIN {X 0,Y 374.375,Z 468.965,A -85,B 0,C 180,E1 -12462.938,E2 -12462.938} C_VEL
LIN {X 0,Y 374.271,Z 470.043,A -85,B 0,C 180,E1 -12464.478,E2 -12464.478} C_VEL
LIN {X 0,Y 374.231,Z 470.305,A -85,B 0,C 180,E1 -12465.988,E2 -12465.988} C_VEL
LIN {X 0,Y 374.21,Z 469.804,A -85,B 0,C 180,E1 -12467.463,E2 -12467.463} C_VEL
LIN {X 0,Y 374.324,Z 468.512,A -85,B 0,C 180,E1 -12468.922,E2 -12468.922} C_VEL
LIN {X 0,Y 374.543,Z 465.256,A -85,B 0,C 180,E1 -12471.056,E2 -12471.056} C_VEL
LIN {X 0,Y 374.744,Z 461.926,A -85,B 0,C 180,E1 -12472.555,E2 -12472.555} C_VEL
LIN {X 0,Y 375.224,Z 456.079,A -85,B 0,C 180,E1 -12474.508,E2 -12474.508} C_VEL
LIN {X 0,Y 375.723,Z 449.571,A -85,B 0,C 180,E1 -12476.19,E2 -12476.19} C_VEL
LIN {X 0,Y 376.376,Z 441.455,A -85,B 0,C 180,E1 -12477.85,E2 -12477.85} C_VEL
LIN {X 0,Y 377.16,Z 432.972,A -85,B 0,C 180,E1 -12479.249,E2 -12479.249} C_VEL
LIN {X 0,Y 378.047,Z 422.577,A -85,B 0,C 180,E1 -12480.642,E2 -12480.642} C_VEL
LIN {X 0,Y 378.96,Z 411.898,A -85,B 0,C 180,E1 -12481.779,E2 -12481.779} C_VEL
LIN {X 0,Y 379.744,Z 400.443,A -85,B 0,C 180,E1 -12482.75,E2 -12482.75} C_VEL
LIN {X 0,Y 380.503,Z 388.317,A -85,B 0,C 180,E1 -12483.541,E2 -12483.541} C_VEL
LIN {X 0,Y 381.093,Z 375.369,A -85,B 0,C 180,E1 -12484.146,E2 -12484.146} C_VEL
LIN {X 0,Y 381.571,Z 361.309,A -85,B 0,C 180,E1 -12484.559,E2 -12484.559} C_VEL
LIN {X 0,Y 382.794,Z 284.179,A -85,B 0,C 180,E1 -12486.107,E2 -12486.107} C_VEL
LIN {X 0,Y 378.399,Z 259.756,A -85,B 0,C 180,E1 -12486.865,E2 -12486.865} C_VEL
LIN {X 0,Y 378.378,Z 258.594,A -85,B 0,C 180,E1 -12487.044,E2 -12487.044} C_VEL
LIN {X 0,Y 378.593,Z 253.985,A -85,B 0,C 180,E1 -12488.208,E2 -12488.208} C_VEL
LIN {X 0,Y 376.343,Z 241.964,A -85,B 0,C 180,E1 -12491.492,E2 -12491.492} C_VEL
LIN {X 0,Y 376.018,Z 240.183,A -85,B 0,C 180,E1 -12492.061,E2 -12492.061} C_VEL
LIN {X 0,Y 375.997,Z 240.147,A -85,B 0,C 180,E1 -12495.939,E2 -12495.939} C_VEL
LIN {X 0,Y 376.021,Z 240.143,A -85,B 0,C 180,E1 -12499.23,E2 -12499.23} C_VEL
LIN {X 0,Y 376.137,Z 240.131,A -85,B 0,C 180,E1 -12502.487,E2 -12502.487} C_VEL
LIN {X 0,Y 376.106,Z 240.136,A -85,B 0,C 180,E1 -12504.641,E2 -12504.641} C_VEL
LIN {X 0,Y 376.286,Z 240.109,A -85,B 0,C 180,E1 -12507.861,E2 -12507.861} C_VEL
LIN {X 0,Y 376.226,Z 240.12,A -85,B 0,C 180,E1 -12508.681,E2 -12508.681} C_VEL
LIN {X 0,Y 375.564,Z 240.211,A -85,B 0,C 180,E1 -12509.574,E2 -12509.574} C_VEL
LIN {X 0,Y 372.747,Z 240.567,A -85,B 0,C 180,E1 -12511.028,E2 -12511.028} C_VEL
LIN {X 0,Y 370.312,Z 240.867,A -85,B 0,C 180,E1 -12512.202,E2 -12512.202} C_VEL
LIN {X 0,Y 369.192,Z 241,A -85,B 0,C 180,E1 -12513.11,E2 -12513.11} C_VEL
LIN {X 0,Y 369.061,Z 241.013,A -85,B 0,C 180,E1 -12513.418,E2 -12513.418} C_VEL
LIN {X 0,Y 369.137,Z 241,A -85,B 0,C 180,E1 -12516.561,E2 -12516.561} C_VEL
LIN {X 0,Y 369.054,Z 241.011,A -85,B 0,C 180,E1 -12518.765,E2 -12518.765} C_VEL
LIN {X 0,Y 368.946,Z 241.024,A -85,B 0,C 180,E1 -12522.097,E2 -12522.097} C_VEL
LIN {X 0,Y 368.932,Z 241.031,A -85,B 0,C 180,E1 -12525.469,E2 -12525.469} C_VEL
LIN {X 0,Y 368.893,Z 241.03,A -85,B 0,C 180,E1 -12528.899,E2 -12528.899} C_VEL
LIN {X 0,Y 368.87,Z 241.034,A -85,B 0,C 180,E1 -12532.401,E2 -12532.401} C_VEL
LIN {X 0,Y 368.941,Z 241.03,A -85,B 0,C 180,E1 -12535.986,E2 -12535.986} C_VEL
LIN {X 0,Y 368.911,Z 241.028,A -85,B 0,C 180,E1 -12538.819,E2 -12538.819} C_VEL
LIN {X 0,Y 368.856,Z 241.04,A -85,B 0,C 180,E1 -12542.244,E2 -12542.244} C_VEL
LIN {X 0,Y 368.878,Z 241.032,A -85,B 0,C 180,E1 -12545.008,E2 -12545.008} C_VEL
LIN {X 0,Y 368.865,Z 241.037,A -85,B 0,C 180,E1 -12548.648,E2 -12548.648} C_VEL
LIN {X 0,Y 368.898,Z 241.032,A -85,B 0,C 180,E1 -12552.027,E2 -12552.027} C_VEL
LIN {X 0,Y 368.95,Z 241.023,A -85,B 0,C 180,E1 -12555.201,E2 -12555.201} C_VEL
LIN {X 0,Y 368.904,Z 241.031,A -85,B 0,C 180,E1 -12558.194,E2 -12558.194} C_VEL
LIN {X 0,Y 368.883,Z 241.032,A -85,B 0,C 180,E1 -12561.367,E2 -12561.367} C_VEL
LIN {X 0,Y 368.908,Z 241.032,A -85,B 0,C 180,E1 -12565.155,E2 -12565.155} C_VEL
LIN {X 0,Y 368.905,Z 241.035,A -85,B 0,C 180,E1 -12569.055,E2 -12569.055} C_VEL
LIN {X 0,Y 368.942,Z 241.027,A -85,B 0,C 180,E1 -12572.805,E2 -12572.805} C_VEL
LIN {X 0,Y 368.917,Z 241.027,A -85,B 0,C 180,E1 -12576.126,E2 -12576.126} C_VEL
LIN {X 0,Y 368.917,Z 241.028,A -85,B 0,C 180,E1 -12579.955,E2 -12579.955} C_VEL
LIN {X 0,Y 368.96,Z 241.028,A -85,B 0,C 180,E1 -12583.407,E2 -12583.407} C_VEL
LIN {X 0,Y 369.053,Z 241.01,A -85,B 0,C 180,E1 -12586.798,E2 -12586.798} C_VEL
LIN {X 0,Y 369.061,Z 241.011,A -85,B 0,C 180,E1 -12590.14,E2 -12590.14} C_VEL
LIN {X 0,Y 369.161,Z 240.999,A -85,B 0,C 180,E1 -12593.449,E2 -12593.449} C_VEL
LIN {X 0,Y 369.312,Z 240.983,A -85,B 0,C 180,E1 -12597.826,E2 -12597.826} C_VEL
LIN {X 0,Y 369.308,Z 240.985,A -85,B 0,C 180,E1 -12602.188,E2 -12602.188} C_VEL
LIN {X 0,Y 369.17,Z 240.999,A -85,B 0,C 180,E1 -12606.566,E2 -12606.566} C_VEL
LIN {X 0,Y 369.073,Z 241.009,A -85,B 0,C 180,E1 -12609.875,E2 -12609.875} C_VEL
LIN {X 0,Y 369.054,Z 241.01,A -85,B 0,C 180,E1 -12613.778,E2 -12613.778} C_VEL
LIN {X 0,Y 369.009,Z 241.015,A -85,B 0,C 180,E1 -12617.748,E2 -12617.748} C_VEL
LIN {X 0,Y 368.929,Z 241.028,A -85,B 0,C 180,E1 -12621.226,E2 -12621.226} C_VEL
LIN {X 0,Y 368.943,Z 241.029,A -85,B 0,C 180,E1 -12624.782,E2 -12624.782} C_VEL
LIN {X 0,Y 368.914,Z 241.031,A -85,B 0,C 180,E1 -12628.796,E2 -12628.796} C_VEL
LIN {X 0,Y 368.919,Z 241.027,A -85,B 0,C 180,E1 -12632.242,E2 -12632.242} C_VEL
LIN {X 0,Y 368.951,Z 241.027,A -85,B 0,C 180,E1 -12635.004,E2 -12635.004} C_VEL
LIN {X 0,Y 368.9,Z 241.029,A -85,B 0,C 180,E1 -12638.637,E2 -12638.637} C_VEL
LIN {X 0,Y 368.877,Z 241.033,A -85,B 0,C 180,E1 -12642.007,E2 -12642.007} C_VEL
LIN {X 0,Y 368.871,Z 241.035,A -85,B 0,C 180,E1 -12645.173,E2 -12645.173} C_VEL
LIN {X 0,Y 368.879,Z 241.033,A -85,B 0,C 180,E1 -12648.175,E2 -12648.175} C_VEL
LIN {X 0,Y 368.899,Z 241.031,A -85,B 0,C 180,E1 -12651.368,E2 -12651.368} C_VEL
LIN {X 0,Y 368.954,Z 241.022,A -85,B 0,C 180,E1 -12655.147,E2 -12655.147} C_VEL
LIN {X 0,Y 368.921,Z 241.029,A -85,B 0,C 180,E1 -12659.044,E2 -12659.044} C_VEL
LIN {X 0,Y 368.961,Z 241.107,A -85,B 0,C 180,E1 -12661.716,E2 -12661.716} C_VEL
LIN {X 0,Y 371.258,Z 252.475,A -85,B 0,C 180,E1 -12664.774,E2 -12664.774} C_VEL
LIN {X 0,Y 372.208,Z 258.62,A -85,B 0,C 180,E1 -12666.343,E2 -12666.343} C_VEL
LIN {X 0,Y 371.288,Z 268.975,A -85,B 0,C 180,E1 -12668.764,E2 -12668.764} C_VEL
LIN {X 0,Y 372.361,Z 275.83,A -85,B 0,C 180,E1 -12669.015,E2 -12669.015} C_VEL
LIN {X 0,Y 376.039,Z 299.17,A -85,B 0,C 180,E1 -12669.703,E2 -12669.703} C_VEL
LIN {X 0,Y 374.577,Z 377.294,A -85,B 0,C 180,E1 -12671.327,E2 -12671.327} C_VEL
LIN {X 0,Y 373.957,Z 390.87,A -85,B 0,C 180,E1 -12671.827,E2 -12671.827} C_VEL
LIN {X 0,Y 373.254,Z 403.768,A -85,B 0,C 180,E1 -12672.536,E2 -12672.536} C_VEL
LIN {X 0,Y 372.311,Z 415.544,A -85,B 0,C 180,E1 -12673.409,E2 -12673.409} C_VEL
LIN {X 0,Y 371.389,Z 426.942,A -85,B 0,C 180,E1 -12674.495,E2 -12674.495} C_VEL
LIN {X 0,Y 370.571,Z 437.227,A -85,B 0,C 180,E1 -12675.725,E2 -12675.725} C_VEL
LIN {X 0,Y 369.699,Z 446.463,A -85,B 0,C 180,E1 -12677.091,E2 -12677.091} C_VEL
LIN {X 0,Y 368.827,Z 455.457,A -85,B 0,C 180,E1 -12678.735,E2 -12678.735} C_VEL
LIN {X 0,Y 368.248,Z 462.67,A -85,B 0,C 180,E1 -12680.385,E2 -12680.385} C_VEL
LIN {X 0,Y 367.897,Z 467.54,A -85,B 0,C 180,E1 -12681.761,E2 -12681.761} C_VEL
LIN {X 0,Y 367.602,Z 472.243,A -85,B 0,C 180,E1 -12683.411,E2 -12683.411} C_VEL
LIN {X 0,Y 367.457,Z 475.809,A -85,B 0,C 180,E1 -12685.061,E2 -12685.061} C_VEL
LIN {X 0,Y 367.361,Z 478.34,A -85,B 0,C 180,E1 -12686.708,E2 -12686.708} C_VEL
LIN {X 0,Y 367.326,Z 479.502,A -85,B 0,C 180,E1 -12687.805,E2 -12687.805} C_VEL
LIN {X 0,Y 367.36,Z 480.22,A -85,B 0,C 180,E1 -12688.902,E2 -12688.902} C_VEL
LIN {X 0,Y 367.384,Z 480.544,A -85,B 0,C 180,E1 -12689.998,E2 -12689.998} C_VEL
LIN {X 0,Y 367.359,Z 480.475,A -85,B 0,C 180,E1 -12691.094,E2 -12691.094} C_VEL
LIN {X 0,Y 367.325,Z 479.988,A -85,B 0,C 180,E1 -12692.191,E2 -12692.191} C_VEL
LIN {X 0,Y 367.362,Z 479.069,A -85,B 0,C 180,E1 -12693.288,E2 -12693.288} C_VEL
LIN {X 0,Y 367.455,Z 477.751,A -85,B 0,C 180,E1 -12694.386,E2 -12694.386} C_VEL
LIN {X 0,Y 367.552,Z 474.851,A -85,B 0,C 180,E1 -12696.092,E2 -12696.092} C_VEL
LIN {X 0,Y 367.838,Z 471.141,A -85,B 0,C 180,E1 -12697.684,E2 -12697.684} C_VEL
LIN {X 0,Y 368.275,Z 466.187,A -85,B 0,C 180,E1 -12699.333,E2 -12699.333} C_VEL
LIN {X 0,Y 368.927,Z 459.953,A -85,B 0,C 180,E1 -12700.98,E2 -12700.98} C_VEL
LIN {X 0,Y 369.753,Z 452.199,A -85,B 0,C 180,E1 -12702.624,E2 -12702.624} C_VEL
LIN {X 0,Y 370.959,Z 442.47,A -85,B 0,C 180,E1 -12704.256,E2 -12704.256} C_VEL
LIN {X 0,Y 371.928,Z 432.461,A -85,B 0,C 180,E1 -12705.619,E2 -12705.619} C_VEL
LIN {X 0,Y 372.926,Z 422.612,A -85,B 0,C 180,E1 -12706.7,E2 -12706.7} C_VEL
LIN {X 0,Y 374.116,Z 410.199,A -85,B 0,C 180,E1 -12707.772,E2 -12707.772} C_VEL
LIN {X 0,Y 374.964,Z 400.314,A -85,B 0,C 180,E1 -12708.437,E2 -12708.437} C_VEL
LIN {X 0,Y 375.761,Z 387.256,A -85,B 0,C 180,E1 -12709.103,E2 -12709.103} C_VEL
LIN {X 0,Y 376.36,Z 374.22,A -85,B 0,C 180,E1 -12709.532,E2 -12709.532} C_VEL
LIN {X 0,Y 378.032,Z 299.534,A -85,B 0,C 180,E1 -12711.102,E2 -12711.102} C_VEL
LIN {X 0,Y 374.512,Z 278.968,A -85,B 0,C 180,E1 -12711.818,E2 -12711.818} C_VEL
LIN {X 0,Y 372.17,Z 268.08,A -85,B 0,C 180,E1 -12712.276,E2 -12712.276} C_VEL
LIN {X 0,Y 372.83,Z 260.937,A -85,B 0,C 180,E1 -12713.907,E2 -12713.907} C_VEL
LIN {X 0,Y 371.714,Z 253.591,A -85,B 0,C 180,E1 -12715.774,E2 -12715.774} C_VEL
LIN {X 0,Y 369.622,Z 243.902,A -85,B 0,C 180,E1 -12718.38,E2 -12718.38} C_VEL
LIN {X 0,Y 368.907,Z 241.068,A -85,B 0,C 180,E1 -12719.253,E2 -12719.253} C_VEL
LIN {X 0,Y 368.909,Z 241.033,A -85,B 0,C 180,E1 -12722.234,E2 -12722.234} C_VEL
LIN {X 0,Y 368.939,Z 241.029,A -85,B 0,C 180,E1 -12724.997,E2 -12724.997} C_VEL
LIN {X 0,Y 368.885,Z 241.034,A -85,B 0,C 180,E1 -12728.629,E2 -12728.629} C_VEL
LIN {X 0,Y 368.866,Z 241.039,A -85,B 0,C 180,E1 -12732,E2 -12732} C_VEL
LIN {X 0,Y 368.878,Z 241.033,A -85,B 0,C 180,E1 -12735.169,E2 -12735.169} C_VEL
LIN {X 0,Y 368.865,Z 241.035,A -85,B 0,C 180,E1 -12738.169,E2 -12738.169} C_VEL
